C07298=1213.014,145.829,-52.403,-178.112,5.931,148.495
C07299=1213.018,145.580,-52.382,-178.114,5.929,148.495
C07300=1213.023,145.331,-52.360,-178.117,5.928,148.496
C07301=1213.027,145.082,-52.340,-178.120,5.927,148.496
C07302=1213.033,144.833,-52.319,-178.122,5.926,148.497
C07303=1213.037,144.584,-52.299,-178.125,5.924,148.497
C07304=1213.042,144.335,-52.278,-178.128,5.922,148.498
C07305=1213.047,144.085,-52.257,-178.130,5.921,148.498
C07306=1213.051,143.837,-52.236,-178.133,5.920,148.499
C07307=1213.056,143.587,-52.214,-178.135,5.919,148.499
C07308=1213.060,143.338,-52.194,-178.138,5.917,148.500
C07309=1213.066,143.089,-52.173,-178.140,5.916,148.500
C07310=1213.070,142.840,-52.153,-178.143,5.915,148.501
C07311=1213.075,142.591,-52.132,-178.145,5.914,148.501
C07312=1213.080,142.342,-52.111,-178.148,5.912,148.502
C07313=1213.084,142.093,-52.091,-178.150,5.911,148.502
C07314=1213.089,141.844,-52.070,-178.153,5.910,148.503
C07315=1213.094,141.595,-52.050,-178.156,5.909,148.503
C07316=1213.099,141.345,-52.029,-178.158,5.907,148.503
C07317=1213.103,141.096,-52.008,-178.161,5.906,148.504
C07318=1213.109,140.847,-51.987,-178.163,5.905,148.504
C07319=1213.113,140.598,-51.967,-178.167,5.903,148.505
C07320=1213.117,140.349,-51.947,-178.169,5.902,148.505
C07321=1213.123,140.100,-51.926,-178.171,5.900,148.506
C07322=1213.127,139.851,-51.905,-178.174,5.900,148.506
C07323=1213.132,139.602,-51.884,-178.177,5.898,148.507
C07324=1213.137,139.353,-51.864,-178.179,5.897,148.507
C07325=1213.141,139.104,-51.844,-178.182,5.896,148.508
C07326=1213.146,138.855,-51.823,-178.184,5.895,148.508
C07327=1213.151,138.606,-51.802,-178.187,5.893,148.509
C07328=1213.156,138.356,-51.781,-178.189,5.892,148.509
C07329=1213.160,138.107,-51.761,-178.192,5.890,148.510
C07330=1213.165,137.859,-51.740,-178.195,5.890,148.510
C07331=1213.170,137.609,-51.720,-178.197,5.888,148.511
C07332=1213.175,137.360,-51.700,-178.200,5.887,148.511
C07333=1213.179,137.111,-51.680,-178.203,5.886,148.512
C07334=1213.184,136.861,-51.659,-178.205,5.885,148.512
C07335=1213.189,136.613,-51.638,-178.208,5.883,148.513
C07336=1213.193,136.364,-51.618,-178.210,5.882,148.513
C07337=1213.198,136.114,-51.597,-178.213,5.881,148.514
C07338=1213.203,135.865,-51.577,-178.215,5.880,148.514
C07339=1213.208,135.616,-51.557,-178.218,5.878,148.514
C07340=1213.212,135.367,-51.536,-178.221,5.877,148.515
C07341=1213.217,135.118,-51.515,-178.223,5.876,148.515
C07342=1213.222,134.869,-51.495,-178.226,5.875,148.516
C07343=1213.226,134.619,-51.475,-178.229,5.873,148.516
C07344=1213.231,134.370,-51.454,-178.231,5.872,148.517
C07345=1213.237,134.122,-51.434,-178.234,5.871,148.517
C07346=1213.241,133.873,-51.414,-178.236,5.870,148.518
C07347=1213.246,133.603,-51.392,-178.239,5.868,148.518
C07348=1213.251,133.335,-51.370,-178.241,5.867,148.519
C07349=1213.256,133.066,-51.349,-178.244,5.866,148.520
C07350=1213.262,132.798,-51.326,-178.248,5.865,148.520
C07351=1213.266,132.548,-51.307,-178.250,5.864,148.521
C07352=1213.271,132.299,-51.286,-178.252,5.862,148.521
C07353=1213.275,132.050,-51.266,-178.255,5.861,148.522
C07354=1213.280,131.801,-51.246,-178.258,5.859,148.522
C07355=1213.286,131.552,-51.226,-178.260,5.859,148.523
C07356=1213.290,131.303,-51.205,-178.263,5.857,148.523
C07357=1213.295,131.054,-51.185,-178.265,5.856,148.524
C07358=1213.299,130.805,-51.165,-178.268,5.855,148.524
C07359=1213.304,130.555,-51.145,-178.270,5.854,148.524
C07360=1213.309,130.306,-51.125,-178.273,5.852,148.525
C07361=1213.314,130.057,-51.104,-178.276,5.851,148.525
C07362=1213.319,129.808,-51.085,-178.278,5.851,148.526
C07363=1213.323,129.559,-51.064,-178.281,5.849,148.526
C07364=1213.328,129.309,-51.045,-178.283,5.848,148.527
C07365=1213.333,129.060,-51.024,-178.286,5.846,148.527
C07366=1213.337,128.811,-51.005,-178.289,5.846,148.528
C07367=1213.342,128.562,-50.984,-178.291,5.844,148.528
C07368=1213.347,128.313,-50.965,-178.294,5.843,148.529
C07369=1213.352,128.064,-50.945,-178.297,5.842,148.529
C07370=1213.357,127.814,-50.924,-178.299,5.841,148.530
C07371=1213.362,127.565,-50.904,-178.301,5.840,148.531
C07372=1213.366,127.316,-50.884,-178.304,5.838,148.531
C07373=1213.371,127.067,-50.864,-178.307,5.838,148.532
C07374=1213.376,126.818,-50.845,-178.309,5.836,148.532
C07375=1213.381,126.569,-50.824,-178.312,5.835,148.533
C07376=1213.385,126.319,-50.805,-178.315,5.833,148.533
C07377=1213.390,126.070,-50.784,-178.317,5.832,148.533
C07378=1213.395,125.822,-50.765,-178.320,5.831,148.534
C07379=1213.399,125.573,-50.745,-178.322,5.830,148.534
C07380=1213.404,125.323,-50.725,-178.325,5.829,148.535
C07381=1213.409,125.073,-50.705,-178.327,5.828,148.535
C07382=1213.414,124.825,-50.685,-178.330,5.827,148.536
C07383=1213.419,124.576,-50.666,-178.333,5.825,148.536
C07384=1213.423,124.326,-50.646,-178.335,5.825,148.537
C07385=1213.428,124.077,-50.626,-178.338,5.823,148.537
C07386=1213.433,123.828,-50.606,-178.341,5.822,148.538
C07387=1213.438,123.579,-50.587,-178.343,5.821,148.539
C07388=1213.442,123.330,-50.566,-178.346,5.820,148.539
C07389=1213.447,123.080,-50.547,-178.348,5.819,148.540
C07390=1213.453,122.831,-50.527,-178.351,5.817,148.540
C07391=1213.457,122.582,-50.507,-178.353,5.817,148.541
C07392=1213.462,122.333,-50.487,-178.355,5.816,148.541
C07393=1213.466,122.083,-50.468,-178.359,5.814,148.542
C07394=1213.471,121.835,-50.448,-178.361,5.813,148.542
C07395=1213.476,121.585,-50.428,-178.364,5.812,148.543
C07396=1213.480,121.336,-50.409,-178.366,5.811,148.543
C07397=1213.486,121.087,-50.390,-178.369,5.809,148.544
C07398=1213.490,120.838,-50.369,-178.371,5.808,148.544
C07399=1213.495,120.589,-50.350,-178.374,5.808,148.545
C07400=1213.500,120.339,-50.330,-178.377,5.806,148.545
C07401=1213.505,120.090,-50.311,-178.379,5.805,148.546
C07402=1213.510,119.841,-50.291,-178.382,5.804,148.546
C07403=1213.514,119.592,-50.271,-178.385,5.803,148.547
C07404=1213.519,119.343,-50.251,-178.387,5.802,148.547
C07405=1213.523,119.094,-50.232,-178.390,5.801,148.548
C07406=1213.528,118.844,-50.213,-178.392,5.800,148.548
C07407=1213.533,118.595,-50.193,-178.395,5.798,148.549
C07408=1213.538,118.346,-50.174,-178.397,5.797,148.549
C07409=1213.544,118.097,-50.155,-178.400,5.797,148.550
C07410=1213.548,117.848,-50.134,-178.403,5.795,148.550
C07411=1213.552,117.599,-50.115,-178.405,5.794,148.551
C07412=1213.557,117.350,-50.096,-178.407,5.793,148.551
C07413=1213.562,117.100,-50.076,-178.410,5.792,148.552
C07414=1213.567,116.851,-50.056,-178.413,5.791,148.552
C07415=1213.572,116.602,-50.037,-178.416,5.789,148.553
C07416=1213.576,116.353,-50.018,-178.418,5.789,148.553
C07417=1213.581,116.103,-49.998,-178.420,5.788,148.554
C07418=1213.586,115.854,-49.979,-178.423,5.786,148.554
C07419=1213.591,115.605,-49.960,-178.426,5.786,148.555
C07420=1213.596,115.356,-49.941,-178.428,5.785,148.555
C07421=1213.600,115.106,-49.921,-178.431,5.783,148.556
C07422=1213.605,114.857,-49.902,-178.433,5.782,148.557
C07423=1213.610,114.608,-49.882,-178.436,5.781,148.557
C07424=1213.614,114.359,-49.863,-178.439,5.780,148.558
C07425=1213.620,114.110,-49.844,-178.441,5.779,148.558
C07426=1213.625,113.860,-49.824,-178.444,5.778,148.559
C07427=1213.630,113.611,-49.805,-178.446,5.777,148.559
C07428=1213.634,113.362,-49.786,-178.449,5.776,148.560
C07429=1213.639,113.113,-49.766,-178.452,5.774,148.560
C07430=1213.644,112.864,-49.747,-178.454,5.774,148.561
C07431=1213.648,112.614,-49.728,-178.456,5.773,148.561
C07432=1213.653,112.366,-49.709,-178.460,5.771,148.562
C07433=1213.658,112.116,-49.689,-178.462,5.771,148.562
C07434=1213.663,111.867,-49.670,-178.464,5.770,148.563
C07435=1213.668,111.617,-49.651,-178.467,5.768,148.563
C07436=1213.673,111.368,-49.632,-178.470,5.768,148.564
C07437=1213.677,111.119,-49.613,-178.472,5.766,148.564
C07438=1213.682,110.870,-49.594,-178.475,5.765,148.565
C07439=1213.687,110.621,-49.574,-178.477,5.764,148.566
C07440=1213.691,110.371,-49.555,-178.480,5.763,148.566
C07441=1213.697,110.123,-49.536,-178.483,5.762,148.567
C07442=1213.702,109.872,-49.517,-178.485,5.761,148.567
C07443=1213.706,109.624,-49.498,-178.488,5.760,148.568
C07444=1213.711,109.374,-49.478,-178.490,5.759,148.568
C07445=1213.716,109.126,-49.460,-178.493,5.758,148.569
C07446=1213.720,108.876,-49.440,-178.496,5.756,148.569
C07447=1213.726,108.627,-49.421,-178.498,5.756,148.570
C07448=1213.730,108.377,-49.402,-178.500,5.755,148.570
C07449=1213.735,108.129,-49.383,-178.504,5.754,148.571
C07450=1213.740,107.880,-49.364,-178.506,5.753,148.572
C07451=1213.745,107.611,-49.344,-178.508,5.752,148.572
C07452=1213.751,107.343,-49.323,-178.511,5.751,148.573
C07453=1213.756,107.073,-49.303,-178.514,5.750,148.573
C07454=1213.761,106.806,-49.283,-178.517,5.749,148.574
C07455=1213.765,106.556,-49.263,-178.519,5.748,148.574
C07456=1213.770,106.307,-49.245,-178.523,5.746,148.575
C07457=1213.775,106.058,-49.225,-178.525,5.745,148.575
C07458=1213.780,105.809,-49.207,-178.527,5.745,148.576
C07459=1213.785,105.559,-49.188,-178.530,5.743,148.576
C07460=1213.789,105.310,-49.169,-178.533,5.742,148.577
C07461=1213.795,105.061,-49.150,-178.535,5.741,148.578
C07462=1213.799,104.812,-49.132,-178.537,5.741,148.578
C07463=1213.804,104.563,-49.112,-178.541,5.739,148.579
C07464=1213.809,104.313,-49.094,-178.543,5.738,148.579
C07465=1213.814,104.064,-49.075,-178.545,5.738,148.580
C07466=1213.818,103.815,-49.056,-178.548,5.736,148.580
C07467=1213.824,103.565,-49.037,-178.551,5.735,148.581
C07468=1213.828,103.317,-49.018,-178.553,5.735,148.582
C07469=1213.833,103.066,-48.999,-178.556,5.733,148.582
C07470=1213.838,102.818,-48.981,-178.558,5.732,148.583
C07471=1213.842,102.568,-48.962,-178.561,5.731,148.583
C07472=1213.847,102.319,-48.943,-178.563,5.731,148.584
C07473=1213.852,102.070,-48.925,-178.566,5.729,148.584
C07474=1213.857,101.820,-48.905,-178.569,5.729,148.585
C07475=1213.862,101.571,-48.887,-178.571,5.728,148.585
C07476=1213.867,101.323,-48.869,-178.574,5.726,148.586
C07477=1213.872,101.072,-48.850,-178.576,5.726,148.586
C07478=1213.876,100.824,-48.831,-178.579,5.725,148.587
C07479=1213.881,100.574,-48.812,-178.581,5.724,148.587
C07480=1213.886,100.325,-48.793,-178.584,5.723,148.588
C07481=1213.891,100.076,-48.775,-178.587,5.722,148.589
C07482=1213.896,99.826,-48.756,-178.589,5.721,148.589
C07483=1213.901,99.577,-48.738,-178.592,5.719,148.590
C07484=1213.905,99.329,-48.719,-178.594,5.719,148.590
C07485=1213.910,99.078,-48.700,-178.597,5.718,148.591
C07486=1213.915,98.829,-48.682,-178.599,5.717,148.591
C07487=1213.920,98.581,-48.663,-178.602,5.716,148.592
C07488=1213.925,98.331,-48.645,-178.605,5.715,148.592
C07489=1213.929,98.082,-48.626,-178.607,5.714,148.593
C07490=1213.934,97.833,-48.608,-178.610,5.713,148.594
C07491=1213.939,97.583,-48.589,-178.612,5.712,148.594
C07492=1213.944,97.334,-48.570,-178.615,5.711,148.595
C07493=1213.949,97.085,-48.552,-178.617,5.710,148.595
C07494=1213.954,96.835,-48.534,-178.620,5.709,148.596
C07495=1213.958,96.586,-48.515,-178.623,5.708,148.596
C07496=1213.963,96.337,-48.497,-178.625,5.707,148.597
C07497=1213.968,96.088,-48.479,-178.628,5.707,148.597
C07498=1213.973,95.838,-48.459,-178.630,5.705,148.598
C07499=1213.978,95.589,-48.441,-178.633,5.704,148.599
C07500=1213.983,95.340,-48.423,-178.636,5.704,148.599
C07501=1213.988,95.091,-48.405,-178.638,5.703,148.600
C07502=1213.993,94.841,-48.385,-178.641,5.702,148.600
C07503=1213.997,94.592,-48.367,-178.644,5.701,148.601
C07504=1214.002,94.343,-48.349,-178.646,5.700,148.601
C07505=1214.007,94.094,-48.331,-178.648,5.699,148.602
C07506=1214.011,93.844,-48.312,-178.651,5.698,148.602
C07507=1214.017,93.595,-48.294,-178.654,5.697,148.603
C07508=1214.022,93.346,-48.276,-178.656,5.696,148.604
C07509=1214.027,93.097,-48.258,-178.658,5.696,148.604
C07510=1214.031,92.847,-48.240,-178.662,5.694,148.605
C07511=1214.036,92.598,-48.221,-178.664,5.694,148.605
C07512=1214.041,92.349,-48.202,-178.666,5.693,148.606
C07513=1214.046,92.099,-48.184,-178.669,5.692,148.606
C07514=1214.051,91.850,-48.166,-178.672,5.690,148.607
C07515=1214.055,91.600,-48.148,-178.674,5.690,148.608
C07516=1214.060,91.351,-48.130,-178.677,5.689,148.608
C07517=1214.065,91.102,-48.112,-178.679,5.688,148.609
C07518=1214.070,90.853,-48.093,-178.682,5.687,148.609
C07519=1214.075,90.603,-48.074,-178.685,5.686,148.610
C07520=1214.080,90.354,-48.056,-178.687,5.685,148.610
C07521=1214.085,90.105,-48.038,-178.690,5.685,148.611
C07522=1214.090,89.856,-48.020,-178.692,5.684,148.612
C07523=1214.095,89.607,-48.002,-178.695,5.682,148.612
C07524=1214.099,89.357,-47.984,-178.698,5.682,148.613
C07525=1214.104,89.108,-47.966,-178.700,5.681,148.613
C07526=1214.109,88.858,-47.948,-178.702,5.680,148.614
C07527=1214.114,88.609,-47.930,-178.706,5.679,148.614
C07528=1214.119,88.360,-47.912,-178.708,5.678,148.615
C07529=1214.123,88.111,-47.894,-178.710,5.677,148.615
C07530=1214.128,87.861,-47.876,-178.713,5.677,148.616
C07531=1214.133,87.611,-47.857,-178.715,5.676,148.617
C07532=1214.138,87.362,-47.839,-178.718,5.674,148.617
C07533=1214.143,87.113,-47.821,-178.721,5.674,148.618
C07534=1214.148,86.864,-47.803,-178.723,5.673,148.618
C07535=1214.153,86.615,-47.785,-178.726,5.672,148.619
C07536=1214.158,86.366,-47.767,-178.728,5.672,148.620
C07537=1214.163,86.116,-47.749,-178.731,5.670,148.620
C07538=1214.167,85.867,-47.731,-178.734,5.669,148.621
C07539=1214.172,85.617,-47.713,-178.736,5.669,148.621
C07540=1214.177,85.368,-47.695,-178.738,5.668,148.622
C07541=1214.182,85.119,-47.677,-178.741,5.667,148.622
C07542=1214.187,84.869,-47.660,-178.744,5.666,148.623
C07543=1214.192,84.620,-47.642,-178.746,5.665,148.623
C07544=1214.197,84.371,-47.624,-178.749,5.664,148.624
C07545=1214.202,84.122,-47.606,-178.752,5.664,148.625
C07546=1214.207,83.873,-47.588,-178.754,5.663,148.625
C07547=1214.210,83.623,-47.570,-178.757,5.661,148.626
C07548=1214.215,83.374,-47.552,-178.759,5.661,148.626
C07549=1214.220,83.125,-47.534,-178.762,5.660,148.627
C07550=1214.225,82.875,-47.517,-178.764,5.659,148.628
C07551=1214.230,82.626,-47.499,-178.767,5.659,148.628
C07552=1214.235,82.376,-47.481,-178.770,5.657,148.629
C07553=1214.240,82.127,-47.463,-178.772,5.656,148.629
C07554=1214.245,81.878,-47.445,-178.775,5.656,148.630
C07555=1214.250,81.609,-47.426,-178.777,5.655,148.631
C07556=1214.256,81.341,-47.407,-178.781,5.654,148.631
C07557=1214.261,81.073,-47.387,-178.783,5.653,148.632
C07558=1214.266,80.804,-47.369,-178.785,5.652,148.632
C07559=1214.271,80.555,-47.351,-178.788,5.652,148.633
C07560=1214.276,80.305,-47.333,-178.791,5.650,148.634
C07561=1214.281,80.056,-47.316,-178.793,5.649,148.634
C07562=1214.285,79.807,-47.298,-178.796,5.649,148.635
C07563=1214.290,79.558,-47.280,-178.799,5.648,148.635
C07564=1214.295,79.308,-47.263,-178.801,5.647,148.636
C07565=1214.300,79.059,-47.245,-178.803,5.647,148.636
C07566=1214.305,78.810,-47.227,-178.807,5.645,148.637
C07567=1214.310,78.560,-47.210,-178.809,5.645,148.638
C07568=1214.315,78.311,-47.192,-178.811,5.644,148.638
C07569=1214.319,78.062,-47.174,-178.814,5.643,148.639
C07570=1214.325,77.812,-47.157,-178.817,5.643,148.640
C07571=1214.330,77.563,-47.139,-178.819,5.642,148.640
C07572=1214.335,77.314,-47.121,-178.822,5.640,148.641
C07573=1214.339,77.064,-47.104,-178.825,5.640,148.641
C07574=1214.344,76.815,-47.086,-178.827,5.639,148.642
C07575=1214.349,76.566,-47.069,-178.829,5.638,148.642
C07576=1214.354,76.316,-47.051,-178.832,5.638,148.643
C07577=1214.358,76.067,-47.034,-178.835,5.637,148.644
C07578=1214.364,75.818,-47.017,-178.837,5.635,148.644
C07579=1214.369,75.569,-46.999,-178.840,5.635,148.645
C07580=1214.374,75.319,-46.982,-178.843,5.634,148.645
C07581=1214.378,75.070,-46.964,-178.845,5.633,148.646
C07582=1214.384,74.820,-46.947,-178.847,5.633,148.646
C07583=1214.388,74.571,-46.929,-178.850,5.632,148.647
C07584=1214.394,74.321,-46.912,-178.852,5.631,148.648
C07585=1214.398,74.072,-46.894,-178.855,5.630,148.648
C07586=1214.403,73.823,-46.877,-178.858,5.629,148.649
C07587=1214.408,73.573,-46.859,-178.861,5.629,148.650
C07588=1214.412,73.324,-46.843,-178.863,5.628,148.650
C07589=1214.417,73.075,-46.825,-178.865,5.627,148.651
C07590=1214.423,72.825,-46.807,-178.868,5.627,148.651
C07591=1214.427,72.576,-46.790,-178.870,5.626,148.652
C07592=1214.432,72.326,-46.773,-178.873,5.625,148.652
C07593=1214.438,72.078,-46.755,-178.876,5.624,148.653
C07594=1214.442,71.828,-46.738,-178.879,5.623,148.654
C07595=1214.447,71.579,-46.720,-178.881,5.622,148.654
C07596=1214.452,71.329,-46.703,-178.883,5.622,148.655
C07597=1214.457,71.080,-46.686,-178.886,5.621,148.655
C07598=1214.462,70.831,-46.668,-178.889,5.620,148.656
C07599=1214.467,70.581,-46.651,-178.891,5.620,148.657
C07600=1214.471,70.332,-46.634,-178.893,5.619,148.657
C07601=1214.477,70.083,-46.617,-178.897,5.618,148.658
C07602=1214.481,69.834,-46.600,-178.899,5.617,148.658
C07603=1214.486,69.584,-46.582,-178.901,5.616,148.659
C07604=1214.491,69.335,-46.565,-178.904,5.616,148.660
C07605=1214.496,69.085,-46.548,-178.907,5.615,148.660
C07606=1214.501,68.836,-46.530,-178.909,5.614,148.661
C07607=1214.505,68.586,-46.514,-178.911,5.613,148.661
C07608=1214.511,68.337,-46.497,-178.914,5.613,148.662
C07609=1214.516,68.088,-46.479,-178.917,5.612,148.663
C07610=1214.520,67.839,-46.462,-178.919,5.611,148.663
C07611=1214.526,67.589,-46.445,-178.922,5.610,148.664
C07612=1214.530,67.339,-46.428,-178.925,5.609,148.664
C07613=1214.535,67.090,-46.410,-178.927,5.609,148.665
C07614=1214.540,66.841,-46.394,-178.929,5.608,148.666
C07615=1214.545,66.592,-46.377,-178.932,5.607,148.666
C07616=1214.550,66.342,-46.360,-178.935,5.607,148.667
C07617=1214.555,66.093,-46.342,-178.937,5.606,148.668
C07618=1214.559,65.844,-46.325,-178.939,5.605,148.668
C07619=1214.564,65.594,-46.308,-178.942,5.605,148.669
C07620=1214.569,65.345,-46.292,-178.945,5.603,148.669
C07621=1214.575,65.095,-46.274,-178.948,5.603,148.670
C07622=1214.579,64.846,-46.257,-178.950,5.602,148.670
C07623=1214.584,64.596,-46.240,-178.953,5.601,148.671
C07624=1214.589,64.348,-46.224,-178.955,5.601,148.672
C07625=1214.594,64.098,-46.206,-178.958,5.600,148.672
C07626=1214.599,63.848,-46.190,-178.960,5.599,148.673
C07627=1214.604,63.599,-46.172,-178.963,5.599,148.673
C07628=1214.608,63.350,-46.155,-178.965,5.598,148.674
C07629=1214.614,63.101,-46.138,-178.968,5.598,148.675
C07630=1214.619,62.851,-46.121,-178.970,5.597,148.675
C07631=1214.623,62.602,-46.105,-178.973,5.596,148.676
C07632=1214.628,62.352,-46.087,-178.976,5.595,148.677
C07633=1214.633,62.103,-46.071,-178.979,5.594,148.677
C07634=1214.639,61.853,-46.054,-178.981,5.593,148.678
C07635=1214.643,61.604,-46.037,-178.983,5.593,148.678
C07636=1214.648,61.355,-46.021,-178.986,5.592,148.679
C07637=1214.653,61.105,-46.004,-178.989,5.592,148.680
C07638=1214.658,60.856,-45.987,-178.991,5.591,148.680
C07639=1214.663,60.606,-45.970,-178.993,5.590,148.681
C07640=1214.668,60.357,-45.953,-178.996,5.590,148.681
C07641=1214.673,60.108,-45.937,-178.999,5.589,148.682
C07642=1214.678,59.858,-45.919,-179.001,5.588,148.682
C07643=1214.682,59.608,-45.903,-179.003,5.588,148.683
C07644=1214.687,59.360,-45.887,-179.006,5.587,148.684
C07645=1214.693,59.110,-45.869,-179.009,5.586,148.684
C07646=1214.697,58.860,-45.853,-179.012,5.585,148.685
C07647=1214.702,58.612,-45.836,-179.014,5.584,148.686
C07648=1214.707,58.362,-45.819,-179.017,5.584,148.686
C07649=1214.712,58.112,-45.802,-179.019,5.583,148.687
C07650=1214.717,57.864,-45.786,-179.022,5.582,148.688
C07651=1214.722,57.614,-45.769,-179.024,5.581,148.688
C07652=1214.727,57.364,-45.752,-179.027,5.581,148.689
C07653=1214.732,57.115,-45.736,-179.029,5.580,148.689
C07654=1214.737,56.866,-45.719,-179.032,5.580,148.690
C07655=1214.741,56.616,-45.702,-179.035,5.579,148.691
C07656=1214.746,56.367,-45.686,-179.037,5.578,148.691
C07657=1214.752,56.118,-45.668,-179.039,5.578,148.692
C07658=1214.757,55.867,-45.652,-179.042,5.577,148.692
C07659=1214.762,55.600,-45.635,-179.045,5.577,148.693
C07660=1214.767,55.332,-45.617,-179.048,5.575,148.694
C07661=1214.773,55.062,-45.599,-179.050,5.575,148.694
C07662=1214.778,54.794,-45.581,-179.053,5.574,148.695
C07663=1214.782,54.545,-45.564,-179.056,5.574,148.696
C07664=1214.788,54.295,-45.547,-179.058,5.573,148.696
C07665=1214.793,54.046,-45.531,-179.061,5.572,148.697
C07666=1214.798,53.796,-45.515,-179.063,5.572,148.698
C07667=1214.803,53.547,-45.499,-179.066,5.571,148.698
C07668=1214.807,53.298,-45.482,-179.068,5.570,148.699
C07669=1214.812,53.048,-45.465,-179.071,5.570,148.699
C07670=1214.817,52.799,-45.448,-179.073,5.569,148.700
C07671=1214.822,52.549,-45.432,-179.076,5.568,148.701
C07672=1214.827,52.301,-45.416,-179.078,5.568,148.701
C07673=1214.832,52.051,-45.400,-179.081,5.567,148.702
C07674=1214.837,51.801,-45.382,-179.083,5.566,148.702
C07675=1214.842,51.552,-45.367,-179.086,5.566,148.703
C07676=1214.847,51.302,-45.350,-179.089,5.565,148.704
C07677=1214.852,51.054,-45.334,-179.091,5.565,148.704
C07678=1214.857,50.803,-45.318,-179.094,5.564,148.705
C07679=1214.862,50.555,-45.301,-179.096,5.563,148.706
C07680=1214.866,50.305,-45.285,-179.099,5.563,148.706
C07681=1214.872,50.055,-45.268,-179.101,5.562,148.707
C07682=1214.877,49.806,-45.252,-179.104,5.562,148.708
C07683=1214.881,49.557,-45.235,-179.106,5.561,148.708
C07684=1214.887,49.307,-45.220,-179.109,5.559,148.709
C07685=1214.891,49.058,-45.203,-179.112,5.559,148.709
C07686=1214.896,48.809,-45.187,-179.114,5.558,148.710
C07687=1214.901,48.559,-45.171,-179.117,5.558,148.711
C07688=1214.906,48.310,-45.154,-179.120,5.557,148.711
C07689=1214.911,48.060,-45.138,-179.122,5.557,148.712
C07690=1214.916,47.811,-45.122,-179.125,5.556,148.712
C07691=1214.920,47.562,-45.105,-179.127,5.555,148.713
C07692=1214.927,47.312,-45.089,-179.130,5.555,148.714
C07693=1214.931,47.062,-45.073,-179.132,5.554,148.714
C07694=1214.936,46.813,-45.057,-179.135,5.554,148.715
C07695=1214.941,46.564,-45.040,-179.137,5.553,148.716
C07696=1214.946,46.315,-45.024,-179.140,5.552,148.716
C07697=1214.951,46.065,-45.008,-179.143,5.552,148.717
C07698=1214.956,45.816,-44.992,-179.145,5.551,148.718
C07699=1214.961,45.566,-44.976,-179.148,5.550,148.718
C07700=1214.966,45.317,-44.960,-179.150,5.550,148.719
C07701=1214.971,45.067,-44.944,-179.153,5.549,148.719
C07702=1214.976,44.818,-44.927,-179.155,5.548,148.720
C07703=1214.980,44.568,-44.911,-179.158,5.548,148.721
C07704=1214.985,44.319,-44.895,-179.161,5.547,148.721
C07705=1214.990,44.069,-44.879,-179.163,5.548,148.722
C07706=1214.996,43.820,-44.864,-179.165,5.547,148.723
C07707=1215.000,43.570,-44.847,-179.167,5.546,148.723
C07708=1215.006,43.321,-44.831,-179.170,5.546,148.724
C07709=1215.010,43.071,-44.815,-179.173,5.545,148.725
C07710=1215.015,42.822,-44.799,-179.175,5.544,148.725
C07711=1215.020,42.573,-44.783,-179.178,5.544,148.726
C07712=1215.025,42.323,-44.767,-179.180,5.543,148.726
C07713=1215.031,42.074,-44.751,-179.183,5.542,148.727
C07714=1215.035,41.824,-44.734,-179.185,5.542,148.728
C07715=1215.040,41.575,-44.719,-179.188,5.541,148.728
C07716=1215.044,41.326,-44.703,-179.191,5.541,148.729
C07717=1215.050,41.076,-44.687,-179.193,5.540,148.730
C07718=1215.055,40.827,-44.672,-179.195,5.539,148.730
C07719=1215.060,40.577,-44.655,-179.198,5.539,148.731
C07720=1215.065,40.328,-44.639,-179.201,5.538,148.731
C07721=1215.070,40.078,-44.623,-179.203,5.538,148.732
C07722=1215.075,39.829,-44.607,-179.206,5.537,148.733
C07723=1215.080,39.580,-44.592,-179.209,5.537,148.734
C07724=1215.085,39.329,-44.576,-179.211,5.536,148.734
C07725=1215.089,39.081,-44.560,-179.213,5.535,148.735
C07726=1215.094,38.831,-44.544,-179.216,5.535,148.735
C07727=1215.099,38.582,-44.528,-179.219,5.534,148.736
C07728=1215.105,38.332,-44.513,-179.221,5.534,148.737
C07729=1215.109,38.083,-44.496,-179.224,5.533,148.737
C07730=1215.115,37.833,-44.480,-179.226,5.532,148.738
C07731=1215.120,37.584,-44.465,-179.229,5.532,148.738
C07732=1215.124,37.335,-44.449,-179.231,5.531,148.739
C07733=1215.129,37.085,-44.433,-179.234,5.531,148.740
C07734=1215.135,36.836,-44.418,-179.237,5.530,148.740
C07735=1215.139,36.586,-44.402,-179.239,5.529,148.741
C07736=1215.145,36.336,-44.386,-179.242,5.529,148.742
C07737=1215.149,36.088,-44.370,-179.244,5.529,148.742
C07738=1215.154,35.838,-44.354,-179.246,5.528,148.743
C07739=1215.159,35.588,-44.339,-179.249,5.528,148.744
C07740=1215.165,35.339,-44.323,-179.251,5.527,148.744
C07741=1215.169,35.089,-44.307,-179.254,5.527,148.745
C07742=1215.174,34.840,-44.292,-179.257,5.526,148.746
C07743=1215.179,34.591,-44.276,-179.259,5.525,148.746
C07744=1215.184,34.341,-44.260,-179.262,5.525,148.747
C07745=1215.189,34.091,-44.244,-179.264,5.524,148.747
C07746=1215.194,33.842,-44.229,-179.267,5.524,148.748
C07747=1215.199,33.592,-44.214,-179.269,5.523,148.749
C07748=1215.204,33.343,-44.198,-179.272,5.523,148.749
C07749=1215.210,33.093,-44.182,-179.275,5.522,148.750
C07750=1215.214,32.844,-44.167,-179.277,5.521,148.751
C07751=1215.219,32.595,-44.151,-179.280,5.521,148.751
C07752=1215.224,32.345,-44.135,-179.282,5.520,148.752
C07753=1215.229,32.096,-44.120,-179.284,5.520,148.753
C07754=1215.234,31.846,-44.104,-179.287,5.520,148.753
C07755=1215.239,31.597,-44.089,-179.290,5.519,148.754
C07756=1215.244,31.347,-44.073,-179.292,5.519,148.755
C07757=1215.248,31.098,-44.058,-179.294,5.518,148.755
C07758=1215.254,30.848,-44.042,-179.297,5.517,148.756
C07759=1215.259,30.599,-44.026,-179.300,5.517,148.756
C07760=1215.264,30.350,-44.011,-179.302,5.516,148.757
C07761=1215.269,30.100,-43.996,-179.305,5.516,148.758
C07762=1215.274,29.850,-43.980,-179.308,5.515,148.758
C07763=1215.279,29.582,-43.964,-179.310,5.515,148.759
C07764=1215.285,29.313,-43.947,-179.313,5.514,148.760
C07765=1215.290,29.045,-43.930,-179.316,5.513,148.761
C07766=1215.295,28.776,-43.914,-179.318,5.513,148.761
C07767=1215.300,28.527,-43.898,-179.321,5.512,148.762
C07768=1215.306,28.276,-43.883,-179.323,5.512,148.763
C07769=1215.310,28.027,-43.868,-179.326,5.511,148.763
C07770=1215.316,27.778,-43.852,-179.329,5.511,148.764
C07771=1215.320,27.529,-43.837,-179.331,5.510,148.764
C07772=1215.325,27.279,-43.821,-179.334,5.509,148.765
C07773=1215.330,27.029,-43.806,-179.336,5.510,148.766
C07774=1215.335,26.780,-43.791,-179.338,5.509,148.766
C07775=1215.340,26.531,-43.775,-179.341,5.509,148.767
C07776=1215.345,26.282,-43.760,-179.344,5.508,148.768
C07777=1215.350,26.032,-43.745,-179.346,5.508,148.768
C07778=1215.356,25.781,-43.729,-179.349,5.507,148.769
C07779=1215.360,25.532,-43.714,-179.351,5.506,148.770
C07780=1215.366,25.283,-43.699,-179.354,5.506,148.770
C07781=1215.370,25.034,-43.684,-179.356,5.505,148.771
C07782=1215.376,24.784,-43.668,-179.359,5.505,148.772
C07783=1215.380,24.535,-43.653,-179.361,5.505,148.772
C07784=1215.385,24.285,-43.638,-179.364,5.504,148.773
C07785=1215.390,24.036,-43.623,-179.366,5.504,148.774
C07786=1215.395,23.786,-43.607,-179.369,5.503,148.774
C07787=1215.400,23.537,-43.592,-179.371,5.502,148.775
C07788=1215.405,23.288,-43.577,-179.374,5.502,148.775
C07789=1215.410,23.038,-43.563,-179.376,5.501,148.776
C07790=1215.415,22.788,-43.547,-179.379,5.501,148.777
C07791=1215.420,22.539,-43.532,-179.382,5.500,148.777
C07792=1215.425,22.289,-43.516,-179.384,5.500,148.778
C07793=1215.430,22.040,-43.502,-179.386,5.500,148.779
C07794=1215.436,21.790,-43.486,-179.389,5.499,148.780
C07795=1215.440,21.541,-43.471,-179.392,5.499,148.780
C07796=1215.446,21.292,-43.456,-179.394,5.498,148.781
C07797=1215.451,21.042,-43.441,-179.396,5.497,148.781
C07798=1215.455,20.792,-43.425,-179.399,5.497,148.782
C07799=1215.460,20.543,-43.410,-179.402,5.496,148.783
C07800=1215.465,20.293,-43.396,-179.404,5.496,148.783
C07801=1215.470,20.044,-43.381,-179.406,5.496,148.784
C07802=1215.475,19.795,-43.366,-179.409,5.496,148.785
C07803=1215.481,19.545,-43.351,-179.412,5.495,148.785
C07804=1215.485,19.296,-43.336,-179.414,5.495,148.786
C07805=1215.491,19.046,-43.320,-179.417,5.494,148.787
C07806=1215.496,18.796,-43.306,-179.419,5.493,148.787
C07807=1215.500,18.547,-43.291,-179.422,5.493,148.788
C07808=1215.506,18.298,-43.275,-179.425,5.492,148.789
C07809=1215.510,18.048,-43.261,-179.427,5.492,148.789
C07810=1215.515,17.798,-43.246,-179.429,5.492,148.790
C07811=1215.520,17.548,-43.231,-179.432,5.491,148.791
C07812=1215.525,17.299,-43.216,-179.435,5.491,148.791
C07813=1215.531,17.049,-43.201,-179.437,5.490,148.792
C07814=1215.535,16.800,-43.186,-179.439,5.489,148.792
C07815=1215.540,16.551,-43.171,-179.442,5.489,148.793
C07816=1215.546,16.301,-43.156,-179.444,5.489,148.794
C07817=1215.550,16.052,-43.141,-179.447,5.489,148.795
C07818=1215.555,15.802,-43.127,-179.449,5.488,148.795
C07819=1215.561,15.553,-43.111,-179.452,5.488,148.796
C07820=1215.566,15.303,-43.097,-179.455,5.487,148.797
C07821=1215.570,15.054,-43.082,-179.457,5.487,148.797
C07822=1215.576,14.804,-43.067,-179.460,5.486,148.798
C07823=1215.581,14.555,-43.052,-179.462,5.486,148.799
C07824=1215.586,14.305,-43.038,-179.464,5.485,148.799
C07825=1215.590,14.056,-43.023,-179.467,5.485,148.800
C07826=1215.596,13.806,-43.008,-179.469,5.484,148.800
C07827=1215.601,13.557,-42.993,-179.472,5.484,148.801
C07828=1215.606,13.307,-42.979,-179.475,5.483,148.802
C07829=1215.611,13.058,-42.963,-179.477,5.483,148.803
C07830=1215.616,12.808,-42.949,-179.479,5.483,148.803
C07831=1215.621,12.559,-42.934,-179.482,5.483,148.804
C07832=1215.625,12.309,-42.919,-179.485,5.482,148.805
C07833=1215.631,12.059,-42.905,-179.487,5.482,148.805
C07834=1215.636,11.810,-42.890,-179.490,5.481,148.806
C07835=1215.641,11.561,-42.875,-179.492,5.480,148.806
C07836=1215.645,11.312,-42.860,-179.494,5.480,148.807
C07837=1215.651,11.061,-42.845,-179.497,5.480,148.808
C07838=1215.656,10.812,-42.831,-179.500,5.479,148.808
C07839=1215.661,10.563,-42.816,-179.502,5.479,148.809
C07840=1215.666,10.313,-42.802,-179.505,5.478,148.810
C07841=1215.671,10.063,-42.788,-179.508,5.478,148.811
C07842=1215.676,9.814,-42.772,-179.510,5.478,148.811
C07843=1215.681,9.564,-42.758,-179.512,5.478,148.812
C07844=1215.686,9.314,-42.743,-179.515,5.477,148.813
C07845=1215.691,9.065,-42.728,-179.517,5.476,148.813
C07846=1215.696,8.816,-42.715,-179.520,5.476,148.814
C07847=1215.702,8.566,-42.700,-179.522,5.475,148.814
C07848=1215.706,8.317,-42.685,-179.524,5.475,148.815
C07849=1215.711,8.068,-42.670,-179.527,5.475,148.816
C07850=1215.716,7.818,-42.656,-179.530,5.474,148.816
C07851=1215.721,7.568,-42.642,-179.532,5.474,148.817
C07852=1215.726,7.319,-42.627,-179.535,5.473,148.818
C07853=1215.731,7.069,-42.613,-179.538,5.473,148.819
C07854=1215.737,6.819,-42.598,-179.540,5.473,148.819
C07855=1215.742,6.570,-42.583,-179.542,5.473,148.820
C07856=1215.746,6.320,-42.568,-179.545,5.472,148.821
C07857=1215.752,6.071,-42.555,-179.547,5.471,148.821
C07858=1215.757,5.822,-42.540,-179.550,5.471,148.822
C07859=1215.762,5.572,-42.526,-179.552,5.471,148.822
C07860=1215.766,5.323,-42.511,-179.555,5.471,148.823
C07861=1215.771,5.073,-42.497,-179.557,5.470,148.824
C07862=1215.776,4.824,-42.482,-179.560,5.470,148.824
C07863=1215.781,4.574,-42.468,-179.563,5.469,148.825
C07864=1215.787,4.324,-42.453,-179.565,5.468,148.826
C07865=1215.792,4.075,-42.439,-179.567,5.469,148.827
C07866=1215.797,3.826,-42.424,-179.570,5.468,148.827
C07867=1215.803,3.556,-42.409,-179.573,5.468,148.828
C07868=1215.808,3.287,-42.394,-179.575,5.467,148.829
C07869=1215.813,3.018,-42.379,-179.578,5.467,148.829
C07870=1215.818,2.749,-42.363,-179.581,5.466,148.830
C07871=1215.823,2.500,-42.349,-179.583,5.466,148.831
C07872=1215.828,2.250,-42.334,-179.586,5.465,148.831
C07873=1215.834,2.001,-42.321,-179.588,5.465,148.832
C07874=1215.839,1.751,-42.306,-179.591,5.465,148.833
C07875=1215.844,1.501,-42.292,-179.593,5.464,148.833
C07876=1215.848,1.252,-42.277,-179.596,5.464,148.834
C07877=1215.853,1.003,-42.263,-179.599,5.463,148.835
C07878=1215.859,0.754,-42.249,-179.601,5.464,148.835
C07879=1215.864,0.504,-42.235,-179.603,5.463,148.836
C07880=1215.869,0.254,-42.220,-179.606,5.463,148.837
C07881=1215.874,0.004,-42.206,-179.608,5.462,148.837
C07882=1215.879,-0.245,-42.192,-179.610,5.462,148.838
C07883=1215.884,-0.494,-42.178,-179.613,5.462,148.839
C07884=1215.889,-0.744,-42.163,-179.616,5.461,148.839
C07885=1215.894,-0.994,-42.149,-179.618,5.461,148.840
C07886=1215.899,-1.243,-42.135,-179.621,5.460,148.841
C07887=1215.904,-1.493,-42.121,-179.623,5.460,148.841
C07888=1215.910,-1.742,-42.107,-179.626,5.460,148.842
C07889=1215.914,-1.992,-42.092,-179.628,5.459,148.843
C07890=1215.919,-2.242,-42.078,-179.631,5.459,148.844
C07891=1215.924,-2.491,-42.064,-179.634,5.458,148.844
C07892=1215.930,-2.740,-42.050,-179.636,5.459,148.845
C07893=1215.935,-2.990,-42.036,-179.638,5.458,148.846
C07894=1215.940,-3.240,-42.021,-179.641,5.458,148.846
C07895=1215.944,-3.490,-42.008,-179.643,5.457,148.847
C07896=1215.950,-3.739,-41.995,-179.645,5.457,148.847
C07897=1215.955,-3.988,-41.980,-179.648,5.457,148.848
C07898=1215.960,-4.238,-41.966,-179.650,5.456,148.849
C07899=1215.965,-4.488,-41.952,-179.653,5.456,148.849
C07900=1215.970,-4.737,-41.938,-179.656,5.455,148.850
C07901=1215.975,-4.987,-41.924,-179.658,5.455,148.851
C07902=1215.980,-5.236,-41.909,-179.660,5.455,148.852
C07903=1215.984,-5.486,-41.896,-179.663,5.454,148.852
C07904=1215.990,-5.735,-41.882,-179.666,5.454,148.853
C07905=1215.995,-5.985,-41.868,-179.668,5.454,148.854
C07906=1216.000,-6.235,-41.854,-179.671,5.454,148.854
C07907=1216.006,-6.484,-41.840,-179.673,5.453,148.855
C07908=1216.011,-6.733,-41.826,-179.676,5.453,148.856
C07909=1216.015,-6.983,-41.812,-179.678,5.453,148.856
C07910=1216.020,-7.233,-41.798,-179.680,5.452,148.857
C07911=1216.026,-7.482,-41.785,-179.683,5.452,148.858
C07912=1216.031,-7.732,-41.770,-179.685,5.451,148.858
C07913=1216.036,-7.982,-41.756,-179.688,5.451,148.859
C07914=1216.041,-8.230,-41.743,-179.690,5.451,148.860
C07915=1216.046,-8.481,-41.729,-179.693,5.450,148.860
C07916=1216.051,-8.730,-41.715,-179.695,5.450,148.861
C07917=1216.056,-8.979,-41.701,-179.698,5.449,148.862
C07918=1216.061,-9.229,-41.687,-179.700,5.450,148.862
C07919=1216.066,-9.479,-41.674,-179.703,5.449,148.863
C07920=1216.071,-9.728,-41.660,-179.705,5.449,148.864
C07921=1216.076,-9.978,-41.645,-179.708,5.448,148.864
C07922=1216.082,-10.228,-41.632,-179.710,5.448,148.865
C07923=1216.086,-10.477,-41.619,-179.713,5.448,148.866
C07924=1216.091,-10.727,-41.604,-179.716,5.447,148.867
C07925=1216.096,-10.976,-41.590,-179.718,5.447,148.867
C07926=1216.102,-11.226,-41.577,-179.720,5.447,148.868
C07927=1216.106,-11.475,-41.563,-179.722,5.446,148.868
C07928=1216.112,-11.724,-41.549,-179.725,5.446,148.869
C07929=1216.117,-11.975,-41.536,-179.728,5.445,148.870
C07930=1216.121,-12.224,-41.522,-179.730,5.446,148.870
C07931=1216.127,-12.473,-41.508,-179.732,5.445,148.871
C07932=1216.132,-12.723,-41.495,-179.735,5.445,148.872
C07933=1216.136,-12.973,-41.481,-179.738,5.444,148.873
C07934=1216.142,-13.222,-41.468,-179.740,5.445,148.873
C07935=1216.147,-13.472,-41.453,-179.743,5.444,148.874
C07936=1216.152,-13.721,-41.440,-179.745,5.444,148.875
C07937=1216.157,-13.971,-41.426,-179.748,5.443,148.875
C07938=1216.162,-14.221,-41.412,-179.750,5.443,148.876
C07939=1216.167,-14.470,-41.400,-179.753,5.443,148.877
C07940=1216.172,-14.720,-41.385,-179.755,5.442,148.877
C07941=1216.178,-14.969,-41.371,-179.757,5.443,148.878
C07942=1216.182,-15.219,-41.358,-179.760,5.442,148.879
C07943=1216.187,-15.469,-41.344,-179.762,5.441,148.879
C07944=1216.193,-15.718,-41.331,-179.765,5.441,148.880
C07945=1216.197,-15.968,-41.317,-179.767,5.441,148.881
C07946=1216.203,-16.217,-41.304,-179.770,5.441,148.881
C07947=1216.208,-16.467,-41.290,-179.772,5.440,148.882
C07948=1216.213,-16.716,-41.277,-179.775,5.440,148.883
C07949=1216.218,-16.966,-41.263,-179.777,5.440,148.883
C07950=1216.223,-17.215,-41.250,-179.780,5.439,148.884
C07951=1216.228,-17.465,-41.236,-179.782,5.439,148.885
C07952=1216.234,-17.715,-41.223,-179.785,5.438,148.885
C07953=1216.238,-17.964,-41.209,-179.787,5.439,148.886
C07954=1216.244,-18.214,-41.196,-179.790,5.438,148.887
C07955=1216.249,-18.463,-41.182,-179.792,5.438,148.888
C07956=1216.254,-18.713,-41.169,-179.794,5.438,148.888
C07957=1216.259,-18.962,-41.155,-179.797,5.438,148.889
C07958=1216.264,-19.212,-41.142,-179.800,5.437,148.890
C07959=1216.270,-19.462,-41.129,-179.802,5.437,148.890
C07960=1216.274,-19.711,-41.115,-179.804,5.437,148.891
C07961=1216.280,-19.961,-41.102,-179.807,5.436,148.892
C07962=1216.284,-20.210,-41.088,-179.809,5.436,148.892
C07963=1216.290,-20.460,-41.075,-179.811,5.436,148.893
C07964=1216.294,-20.710,-41.062,-179.814,5.435,148.894
C07965=1216.300,-20.959,-41.048,-179.817,5.435,148.894
C07966=1216.305,-21.209,-41.035,-179.819,5.434,148.895
C07967=1216.310,-21.458,-41.021,-179.821,5.435,148.896
C07968=1216.315,-21.708,-41.008,-179.824,5.434,148.896
C07969=1216.320,-21.958,-40.995,-179.827,5.434,148.897
C07970=1216.325,-22.207,-40.981,-179.829,5.434,148.898
C07971=1216.331,-22.477,-40.967,-179.831,5.434,148.898
C07972=1216.336,-22.746,-40.952,-179.834,5.433,148.899
C07973=1216.341,-23.016,-40.939,-179.837,5.433,148.900
C07974=1216.347,-23.285,-40.924,-179.840,5.432,148.901
C07975=1216.352,-23.534,-40.911,-179.842,5.433,148.901
C07976=1216.358,-23.784,-40.898,-179.845,5.432,148.902
C07977=1216.362,-24.033,-40.884,-179.847,5.432,148.903
C07978=1216.368,-24.283,-40.871,-179.850,5.431,148.904
C07979=1216.372,-24.533,-40.858,-179.852,5.431,148.904
C07980=1216.378,-24.783,-40.845,-179.854,5.431,148.905
C07981=1216.383,-25.032,-40.831,-179.857,5.430,148.905
C07982=1216.388,-25.281,-40.819,-179.859,5.431,148.906
C07983=1216.393,-25.532,-40.805,-179.862,5.430,148.907
C07984=1216.398,-25.781,-40.792,-179.864,5.430,148.908
C07985=1216.403,-26.031,-40.778,-179.866,5.430,148.908
C07986=1216.408,-26.280,-40.766,-179.869,5.429,148.909
C07987=1216.413,-26.529,-40.753,-179.872,5.429,148.910
C07988=1216.419,-26.780,-40.739,-179.874,5.428,148.910
C07989=1216.423,-27.028,-40.726,-179.876,5.429,148.911
C07990=1216.429,-27.279,-40.713,-179.879,5.428,148.912
C07991=1216.434,-27.528,-40.700,-179.882,5.428,148.912
C07992=1216.439,-27.777,-40.687,-179.884,5.428,148.913
C07993=1216.444,-28.028,-40.674,-179.886,5.428,148.914
C07994=1216.449,-28.277,-40.661,-179.889,5.427,148.914
C07995=1216.453,-28.526,-40.647,-179.891,5.427,148.915
C07996=1216.459,-28.776,-40.634,-179.894,5.427,148.916
C07997=1216.464,-29.025,-40.622,-179.897,5.427,148.917
C07998=1216.469,-29.275,-40.609,-179.898,5.426,148.917
C07999=1216.475,-29.525,-40.596,-179.901,5.426,148.918
C08000=1216.479,-29.775,-40.583,-179.903,5.425,148.918
C08001=1216.484,-30.024,-40.570,-179.906,5.426,148.919
C08002=1216.490,-30.274,-40.557,-179.908,5.425,148.920
C08003=1216.495,-30.523,-40.543,-179.911,5.425,148.921
C08004=1216.500,-30.773,-40.530,-179.914,5.424,148.921
C08005=1216.506,-31.022,-40.517,-179.916,5.425,148.922
C08006=1216.510,-31.272,-40.504,-179.918,5.424,148.923
C08007=1216.515,-31.522,-40.492,-179.921,5.424,148.923
C08008=1216.521,-31.771,-40.479,-179.923,5.424,148.924
C08009=1216.526,-32.021,-40.466,-179.926,5.424,148.925
C08010=1216.531,-32.271,-40.453,-179.928,5.423,148.925
C08011=1216.536,-32.520,-40.440,-179.930,5.423,148.926
C08012=1216.541,-32.770,-40.427,-179.933,5.423,148.927
C08013=1216.546,-33.020,-40.414,-179.936,5.422,148.928
C08014=1216.551,-33.269,-40.402,-179.938,5.423,148.928
C08015=1216.556,-33.519,-40.389,-179.940,5.422,148.929
C08016=1216.562,-33.769,-40.375,-179.943,5.422,148.930
C08017=1216.567,-34.018,-40.363,-179.945,5.422,148.930
C08018=1216.571,-34.268,-40.350,-179.947,5.421,148.931
C08019=1216.576,-34.517,-40.337,-179.950,5.421,148.931
C08020=1216.582,-34.767,-40.324,-179.952,5.421,148.932
C08021=1216.587,-35.017,-40.311,-179.955,5.421,148.933
C08022=1216.592,-35.266,-40.299,-179.957,5.420,148.934
C08023=1216.597,-35.516,-40.286,-179.960,5.420,148.934
C08024=1216.602,-35.765,-40.273,-179.962,5.420,148.935
C08025=1216.607,-36.015,-40.260,-179.965,5.419,148.936
C08026=1216.613,-36.264,-40.247,-179.967,5.420,148.936
C08027=1216.618,-36.514,-40.235,-179.970,5.419,148.937
C08028=1216.623,-36.763,-40.222,-179.972,5.419,148.938
C08029=1216.628,-37.014,-40.210,-179.974,5.419,148.938
C08030=1216.634,-37.263,-40.196,-179.977,5.419,148.939
C08031=1216.639,-37.513,-40.184,-179.980,5.418,148.940
C08032=1216.643,-37.763,-40.171,-179.982,5.419,148.941
C08033=1216.648,-38.012,-40.158,-179.984,5.418,148.941
C08034=1216.653,-38.261,-40.146,-179.987,5.418,148.942
C08035=1216.659,-38.511,-40.133,-179.989,5.418,148.943
C08036=1216.664,-38.761,-40.120,-179.992,5.417,148.943
C08037=1216.669,-39.011,-40.108,-179.994,5.418,148.944
C08038=1216.674,-39.260,-40.095,-179.996,5.417,148.945
C08039=1216.680,-39.510,-40.082,-179.999,5.416,148.945
C08040=1216.685,-39.759,-40.070,179.999,5.417,148.946
C08041=1216.689,-40.009,-40.057,179.997,5.416,148.947
C08042=1216.695,-40.259,-40.045,179.994,5.416,148.947
C08043=1216.700,-40.508,-40.032,179.992,5.416,148.948
C08044=1216.705,-40.757,-40.020,179.989,5.416,148.949
C08045=1216.709,-41.008,-40.007,179.986,5.415,148.949
C08046=1216.715,-41.257,-39.994,179.984,5.416,148.950
C08047=1216.721,-41.507,-39.982,179.982,5.415,148.951
C08048=1216.726,-41.756,-39.969,179.979,5.415,148.952
C08049=1216.731,-42.006,-39.957,179.977,5.415,148.952
C08050=1216.735,-42.256,-39.944,179.974,5.414,148.953
C08051=1216.741,-42.506,-39.932,179.972,5.414,148.954
C08052=1216.746,-42.755,-39.919,179.970,5.414,148.954
C08053=1216.751,-43.004,-39.907,179.967,5.414,148.955
C08054=1216.756,-43.254,-39.894,179.965,5.414,148.956
C08055=1216.761,-43.504,-39.882,179.962,5.414,148.956
C08056=1216.766,-43.754,-39.869,179.959,5.413,148.957
C08057=1216.771,-44.003,-39.856,179.957,5.414,148.958
C08058=1216.777,-44.253,-39.845,179.955,5.413,148.958
C08059=1216.782,-44.502,-39.832,179.953,5.412,148.959
C08060=1216.787,-44.751,-39.819,179.950,5.413,148.960
C08061=1216.792,-45.002,-39.807,179.948,5.412,148.960
C08062=1216.797,-45.251,-39.795,179.945,5.412,148.961
C08063=1216.802,-45.501,-39.782,179.943,5.412,148.962
C08064=1216.807,-45.751,-39.770,179.940,5.411,148.963
C08065=1216.813,-46.000,-39.757,179.938,5.412,148.963
C08066=1216.818,-46.249,-39.745,179.936,5.411,148.964
C08067=1216.823,-46.499,-39.733,179.933,5.411,148.965
C08068=1216.828,-46.749,-39.720,179.931,5.411,148.965
C08069=1216.833,-46.999,-39.708,179.928,5.411,148.966
C08070=1216.838,-47.249,-39.696,179.926,5.410,148.967
C08071=1216.843,-47.498,-39.683,179.923,5.411,148.967
C08072=1216.849,-47.748,-39.671,179.921,5.410,148.968
C08073=1216.854,-47.997,-39.658,179.919,5.410,148.969
C08074=1216.859,-48.247,-39.647,179.916,5.410,148.970
C08075=1216.864,-48.517,-39.633,179.913,5.410,148.970
C08076=1216.870,-48.787,-39.620,179.911,5.409,148.971
C08077=1216.876,-49.056,-39.606,179.909,5.409,148.972
C08078=1216.881,-49.327,-39.593,179.906,5.409,148.972
C08079=1216.886,-49.576,-39.580,179.903,5.408,148.973
C08080=1216.892,-49.826,-39.569,179.901,5.409,148.974
C08081=1216.896,-50.075,-39.557,179.899,5.408,148.974
C08082=1216.902,-50.325,-39.545,179.896,5.408,148.975
C08083=1216.907,-50.574,-39.532,179.894,5.408,148.976
C08084=1216.912,-50.824,-39.520,179.891,5.408,148.977
C08085=1216.917,-51.074,-39.508,179.889,5.408,148.977
C08086=1216.922,-51.324,-39.495,179.886,5.408,148.978
C08087=1216.927,-51.574,-39.483,179.884,5.407,148.979
C08088=1216.933,-51.823,-39.471,179.882,5.407,148.979
C08089=1216.937,-52.073,-39.460,179.879,5.407,148.980
C08090=1216.943,-52.322,-39.447,179.877,5.407,148.981
C08091=1216.948,-52.572,-39.435,179.874,5.407,148.982
C08092=1216.953,-52.822,-39.422,179.872,5.406,148.982
C08093=1216.959,-53.072,-39.411,179.870,5.406,148.983
C08094=1216.964,-53.321,-39.398,179.867,5.406,148.983
C08095=1216.968,-53.571,-39.387,179.865,5.406,148.984
C08096=1216.973,-53.820,-39.374,179.863,5.406,148.985
C08097=1216.979,-54.070,-39.362,179.860,5.405,148.986
C08098=1216.984,-54.320,-39.350,179.858,5.406,148.986
C08099=1216.989,-54.569,-39.338,179.855,5.405,148.987
C08100=1216.994,-54.819,-39.326,179.852,5.405,148.988
C08101=1217.000,-55.069,-39.315,179.850,5.405,148.988
C08102=1217.005,-55.318,-39.302,179.848,5.405,148.989
C08103=1217.010,-55.568,-39.290,179.846,5.405,148.990
C08104=1217.015,-55.817,-39.277,179.843,5.404,148.990
C08105=1217.020,-56.067,-39.266,179.840,5.404,148.991
C08106=1217.025,-56.317,-39.254,179.838,5.404,148.992
C08107=1217.030,-56.566,-39.242,179.836,5.404,148.993
C08108=1217.036,-56.816,-39.230,179.833,5.404,148.993
C08109=1217.041,-57.066,-39.218,179.831,5.404,148.994
C08110=1217.046,-57.315,-39.206,179.829,5.403,148.994
C08111=1217.051,-57.565,-39.194,179.827,5.403,148.995
C08112=1217.057,-57.815,-39.182,179.824,5.403,148.996
C08113=1217.061,-58.064,-39.171,179.822,5.403,148.997
C08114=1217.066,-58.314,-39.158,179.819,5.403,148.997
C08115=1217.072,-58.564,-39.146,179.817,5.403,148.998
C08116=1217.077,-58.813,-39.135,179.814,5.403,148.999
C08117=1217.082,-59.063,-39.123,179.812,5.402,148.999
C08118=1217.087,-59.313,-39.111,179.810,5.402,149.000
C08119=1217.093,-59.563,-39.099,179.807,5.402,149.001
C08120=1217.097,-59.812,-39.087,179.805,5.402,149.001
C08121=1217.103,-60.062,-39.075,179.802,5.402,149.002
C08122=1217.108,-60.311,-39.063,179.799,5.401,149.003
C08123=1217.112,-60.561,-39.052,179.797,5.402,149.004
C08124=1217.118,-60.811,-39.040,179.795,5.401,149.004
C08125=1217.123,-61.061,-39.028,179.793,5.401,149.005
C08126=1217.128,-61.310,-39.016,179.790,5.401,149.005
C08127=1217.133,-61.560,-39.004,179.788,5.400,149.006
C08128=1217.139,-61.810,-38.992,179.786,5.401,149.007
C08129=1217.143,-62.059,-38.981,179.783,5.400,149.008
C08130=1217.149,-62.309,-38.969,179.781,5.401,149.008
C08131=1217.155,-62.559,-38.957,179.778,5.400,149.009
C08132=1217.159,-62.808,-38.945,179.776,5.400,149.010
C08133=1217.165,-63.058,-38.933,179.774,5.400,149.010
C08134=1217.169,-63.307,-38.922,179.771,5.400,149.011
C08135=1217.175,-63.557,-38.910,179.769,5.400,149.012
C08136=1217.180,-63.807,-38.898,179.766,5.399,149.013
C08137=1217.185,-64.057,-38.887,179.764,5.400,149.013
C08138=1217.190,-64.307,-38.875,179.761,5.399,149.014
C08139=1217.196,-64.557,-38.863,179.759,5.399,149.014
C08140=1217.200,-64.806,-38.852,179.757,5.399,149.015
C08141=1217.206,-65.055,-38.840,179.754,5.398,149.016
C08142=1217.211,-65.304,-38.829,179.752,5.399,149.017
C08143=1217.216,-65.554,-38.817,179.750,5.398,149.017
C08144=1217.221,-65.804,-38.805,179.748,5.399,149.018
C08145=1217.226,-66.054,-38.793,179.745,5.398,149.019
C08146=1217.232,-66.304,-38.782,179.742,5.398,149.019
C08147=1217.236,-66.553,-38.770,179.740,5.398,149.020
C08148=1217.242,-66.803,-38.758,179.737,5.398,149.021
C08149=1217.247,-67.052,-38.747,179.735,5.398,149.022
C08150=1217.253,-67.302,-38.736,179.733,5.398,149.022
C08151=1217.257,-67.552,-38.724,179.731,5.398,149.023
C08152=1217.263,-67.802,-38.712,179.728,5.397,149.024
C08153=1217.267,-68.051,-38.701,179.726,5.397,149.024
C08154=1217.273,-68.301,-38.689,179.724,5.397,149.025
C08155=1217.278,-68.550,-38.678,179.721,5.396,149.026
C08156=1217.284,-68.800,-38.666,179.719,5.397,149.026
C08157=1217.288,-69.050,-38.655,179.716,5.396,149.027
C08158=1217.294,-69.300,-38.643,179.714,5.397,149.028
C08159=1217.298,-69.549,-38.632,179.712,5.396,149.028
C08160=1217.304,-69.799,-38.620,179.709,5.397,149.029
C08161=1217.309,-70.048,-38.609,179.707,5.396,149.030
C08162=1217.314,-70.298,-38.597,179.704,5.396,149.030
C08163=1217.319,-70.548,-38.586,179.702,5.396,149.031
C08164=1217.325,-70.798,-38.574,179.699,5.396,149.032
C08165=1217.330,-71.048,-38.564,179.698,5.396,149.032
C08166=1217.336,-71.297,-38.552,179.695,5.395,149.033
C08167=1217.340,-71.547,-38.541,179.693,5.395,149.034
C08168=1217.346,-71.797,-38.529,179.690,5.395,149.034
C08169=1217.350,-72.046,-38.518,179.688,5.395,149.035
C08170=1217.356,-72.296,-38.506,179.686,5.395,149.036
C08171=1217.361,-72.545,-38.495,179.683,5.394,149.037
C08172=1217.367,-72.795,-38.483,179.681,5.395,149.037
C08173=1217.371,-73.045,-38.472,179.678,5.394,149.038
C08174=1217.376,-73.295,-38.461,179.676,5.395,149.039
C08175=1217.382,-73.544,-38.449,179.673,5.394,149.039
C08176=1217.387,-73.794,-38.438,179.671,5.395,149.040
C08177=1217.392,-74.044,-38.426,179.669,5.394,149.041
C08178=1217.397,-74.294,-38.415,179.667,5.394,149.041
C08179=1217.403,-74.564,-38.403,179.664,5.394,149.042
C08180=1217.409,-74.835,-38.391,179.661,5.394,149.043
C08181=1217.414,-75.105,-38.378,179.659,5.393,149.044
C08182=1217.420,-75.375,-38.366,179.656,5.394,149.044
C08183=1217.425,-75.625,-38.355,179.654,5.393,149.045
C08184=1217.430,-75.875,-38.344,179.652,5.393,149.046
C08185=1217.436,-76.125,-38.333,179.649,5.393,149.047
C08186=1217.441,-76.374,-38.321,179.647,5.393,149.047
C08187=1217.446,-76.624,-38.310,179.644,5.393,149.048
C08188=1217.452,-76.874,-38.299,179.643,5.393,149.048
C08189=1217.457,-77.123,-38.288,179.640,5.392,149.049
C08190=1217.461,-77.373,-38.277,179.637,5.392,149.050
C08191=1217.467,-77.623,-38.265,179.635,5.392,149.051
C08192=1217.472,-77.872,-38.255,179.633,5.392,149.051
C08193=1217.477,-78.122,-38.243,179.630,5.392,149.052
C08194=1217.482,-78.372,-38.231,179.628,5.392,149.053
C08195=1217.488,-78.621,-38.220,179.626,5.392,149.053
C08196=1217.493,-78.871,-38.210,179.623,5.392,149.054
C08197=1217.498,-79.121,-38.198,179.621,5.392,149.055
C08198=1217.503,-79.371,-38.187,179.619,5.391,149.055
C08199=1217.508,-79.620,-38.177,179.617,5.392,149.056
C08200=1217.514,-79.870,-38.165,179.614,5.391,149.057
C08201=1217.519,-80.120,-38.153,179.611,5.391,149.057
C08202=1217.524,-80.369,-38.143,179.609,5.391,149.058
C08203=1217.529,-80.619,-38.132,179.607,5.391,149.059
C08204=1217.534,-80.869,-38.120,179.604,5.391,149.060
C08205=1217.540,-81.118,-38.110,179.602,5.391,149.060
C08206=1217.545,-81.368,-38.098,179.600,5.391,149.061
C08207=1217.550,-81.619,-38.087,179.597,5.391,149.062
C08208=1217.556,-81.868,-38.076,179.595,5.390,149.062
C08209=1217.560,-82.117,-38.065,179.593,5.390,149.063
C08210=1217.565,-82.367,-38.055,179.591,5.390,149.064
C08211=1217.571,-82.616,-38.044,179.588,5.390,149.064
C08212=1217.576,-82.867,-38.032,179.586,5.390,149.065
C08213=1217.582,-83.116,-38.021,179.583,5.390,149.066
C08214=1217.586,-83.365,-38.010,179.581,5.390,149.066
C08215=1217.591,-83.616,-38.000,179.578,5.390,149.067
C08216=1217.597,-83.865,-37.988,179.576,5.389,149.068
C08217=1217.602,-84.115,-37.978,179.574,5.390,149.069
C08218=1217.607,-84.365,-37.966,179.572,5.389,149.069
C08219=1217.613,-84.614,-37.956,179.569,5.389,149.070
C08220=1217.617,-84.864,-37.945,179.567,5.389,149.070
C08221=1217.623,-85.114,-37.934,179.565,5.389,149.071
C08222=1217.628,-85.363,-37.923,179.562,5.389,149.072
C08223=1217.633,-85.614,-37.912,179.560,5.389,149.073
C08224=1217.639,-85.863,-37.901,179.557,5.389,149.073
C08225=1217.644,-86.113,-37.891,179.555,5.389,149.074
C08226=1217.648,-86.362,-37.879,179.552,5.389,149.075
C08227=1217.654,-86.612,-37.869,179.551,5.389,149.075
C08228=1217.659,-86.862,-37.857,179.548,5.388,149.076
C08229=1217.665,-87.111,-37.847,179.546,5.388,149.077
C08230=1217.670,-87.361,-37.836,179.543,5.388,149.077
C08231=1217.675,-87.611,-37.825,179.541,5.388,149.078
C08232=1217.680,-87.860,-37.814,179.539,5.388,149.079
C08233=1217.685,-88.111,-37.804,179.537,5.388,149.079
C08234=1217.690,-88.359,-37.793,179.534,5.388,149.080
C08235=1217.696,-88.610,-37.782,179.532,5.388,149.081
C08236=1217.701,-88.859,-37.771,179.530,5.387,149.081
C08237=1217.706,-89.109,-37.760,179.528,5.388,149.082
C08238=1217.712,-89.359,-37.750,179.525,5.387,149.083
C08239=1217.717,-89.608,-37.739,179.522,5.387,149.083
C08240=1217.722,-89.859,-37.728,179.520,5.387,149.084
C08241=1217.727,-90.107,-37.717,179.517,5.387,149.085
C08242=1217.732,-90.358,-37.706,179.515,5.387,149.086
C08243=1217.737,-90.607,-37.696,179.513,5.387,149.086
C08244=1217.742,-90.857,-37.685,179.511,5.387,149.087
C08245=1217.748,-91.106,-37.675,179.508,5.386,149.088
C08246=1217.753,-91.357,-37.664,179.506,5.387,149.088
C08247=1217.759,-91.606,-37.653,179.504,5.386,149.089
C08248=1217.764,-91.856,-37.642,179.502,5.387,149.090
C08249=1217.769,-92.106,-37.632,179.499,5.386,149.090
C08250=1217.774,-92.355,-37.621,179.497,5.387,149.091
C08251=1217.780,-92.605,-37.610,179.495,5.386,149.092
C08252=1217.785,-92.855,-37.600,179.493,5.386,149.092
C08253=1217.790,-93.104,-37.589,179.490,5.386,149.093
C08254=1217.795,-93.354,-37.578,179.488,5.386,149.094
C08255=1217.801,-93.604,-37.568,179.485,5.386,149.094
C08256=1217.806,-93.854,-37.558,179.483,5.386,149.095
C08257=1217.811,-94.103,-37.547,179.480,5.386,149.096
C08258=1217.816,-94.353,-37.536,179.478,5.386,149.097
C08259=1217.821,-94.603,-37.526,179.476,5.385,149.097
C08260=1217.826,-94.852,-37.515,179.474,5.385,149.098
C08261=1217.832,-95.102,-37.504,179.471,5.385,149.098
C08262=1217.837,-95.352,-37.494,179.469,5.385,149.099
C08263=1217.842,-95.602,-37.484,179.467,5.385,149.100
C08264=1217.847,-95.852,-37.473,179.464,5.385,149.101
C08265=1217.853,-96.101,-37.462,179.462,5.385,149.101
C08266=1217.858,-96.351,-37.451,179.460,5.385,149.102
C08267=1217.863,-96.601,-37.441,179.457,5.384,149.102
C08268=1217.868,-96.851,-37.431,179.455,5.385,149.103
C08269=1217.873,-97.100,-37.420,179.453,5.384,149.104
C08270=1217.879,-97.349,-37.410,179.451,5.385,149.105
C08271=1217.884,-97.600,-37.399,179.448,5.384,149.105
C08272=1217.889,-97.849,-37.389,179.446,5.385,149.106
C08273=1217.894,-98.099,-37.379,179.444,5.384,149.107
C08274=1217.900,-98.349,-37.369,179.442,5.384,149.107
C08275=1217.904,-98.598,-37.357,179.439,5.384,149.108
C08276=1217.910,-98.848,-37.347,179.437,5.384,149.109
C08277=1217.915,-99.098,-37.336,179.434,5.384,149.109
C08278=1217.920,-99.348,-37.326,179.432,5.384,149.110
C08279=1217.926,-99.597,-37.316,179.429,5.384,149.111
C08280=1217.931,-99.847,-37.305,179.428,5.384,149.111
C08281=1217.937,-100.097,-37.295,179.425,5.383,149.112
C08282=1217.942,-100.347,-37.285,179.423,5.384,149.113
C08283=1217.947,-100.617,-37.273,179.420,5.383,149.113
C08284=1217.952,-100.888,-37.262,179.418,5.384,149.114
C08285=1217.958,-101.160,-37.251,179.416,5.383,149.115
C08286=1217.964,-101.431,-37.240,179.413,5.383,149.116
C08287=1217.969,-101.681,-37.230,179.411,5.383,149.116
C08288=1217.975,-101.930,-37.220,179.408,5.383,149.117
C08289=1217.980,-102.181,-37.209,179.406,5.383,149.118
C08290=1217.985,-102.430,-37.199,179.403,5.383,149.118
C08291=1217.991,-102.680,-37.189,179.401,5.383,149.119
C08292=1217.995,-102.930,-37.179,179.399,5.383,149.120
C08293=1218.001,-103.179,-37.168,179.397,5.383,149.120
C08294=1218.006,-103.430,-37.158,179.394,5.382,149.121
C08295=1218.011,-103.679,-37.148,179.392,5.383,149.122
C08296=1218.017,-103.929,-37.137,179.390,5.382,149.122
C08297=1218.022,-104.178,-37.126,179.387,5.382,149.123
C08298=1218.026,-104.427,-37.117,179.385,5.382,149.124
C08299=1218.032,-104.678,-37.107,179.383,5.382,149.124
C08300=1218.037,-104.928,-37.096,179.381,5.382,149.125
C08301=1218.043,-105.177,-37.086,179.378,5.382,149.126
C08302=1218.048,-105.427,-37.076,179.376,5.382,149.127
C08303=1218.053,-105.677,-37.066,179.374,5.382,149.127
C08304=1218.058,-105.926,-37.056,179.372,5.382,149.128
C08305=1218.064,-106.176,-37.046,179.369,5.382,149.128
C08306=1218.069,-106.426,-37.035,179.367,5.382,149.129
C08307=1218.074,-106.675,-37.025,179.365,5.381,149.130
C08308=1218.079,-106.925,-37.015,179.363,5.382,149.131
C08309=1218.084,-107.175,-37.005,179.360,5.381,149.131
C08310=1218.090,-107.425,-36.994,179.358,5.382,149.132
C08311=1218.095,-107.674,-36.985,179.356,5.381,149.133
C08312=1218.100,-107.924,-36.974,179.353,5.381,149.133
C08313=1218.105,-108.174,-36.964,179.351,5.381,149.134
C08314=1218.111,-108.423,-36.954,179.349,5.381,149.135
C08315=1218.116,-108.674,-36.945,179.346,5.381,149.135
C08316=1218.121,-108.923,-36.934,179.344,5.381,149.136
C08317=1218.127,-109.173,-36.924,179.342,5.380,149.137
C08318=1218.131,-109.423,-36.914,179.340,5.381,149.137
C08319=1218.137,-109.672,-36.904,179.337,5.380,149.138
C08320=1218.142,-109.922,-36.894,179.335,5.381,149.139
C08321=1218.148,-110.172,-36.884,179.332,5.380,149.139
C08322=1218.152,-110.422,-36.874,179.331,5.380,149.140
C08323=1218.158,-110.672,-36.864,179.328,5.380,149.141
C08324=1218.164,-110.921,-36.854,179.326,5.380,149.141
C08325=1218.168,-111.170,-36.844,179.324,5.381,149.142
C08326=1218.173,-111.421,-36.834,179.321,5.380,149.143
C08327=1218.179,-111.670,-36.823,179.319,5.380,149.143
C08328=1218.184,-111.920,-36.815,179.317,5.380,149.144
C08329=1218.190,-112.170,-36.804,179.315,5.380,149.145
C08330=1218.195,-112.420,-36.794,179.312,5.380,149.145
C08331=1218.200,-112.669,-36.784,179.310,5.380,149.146
C08332=1218.206,-112.919,-36.775,179.308,5.379,149.147
C08333=1218.211,-113.169,-36.764,179.306,5.380,149.147
C08334=1218.215,-113.419,-36.755,179.303,5.379,149.148
C08335=1218.221,-113.668,-36.744,179.301,5.380,149.149
C08336=1218.226,-113.918,-36.735,179.298,5.379,149.149
C08337=1218.232,-114.168,-36.725,179.297,5.379,149.150
C08338=1218.237,-114.418,-36.715,179.294,5.379,149.151
C08339=1218.242,-114.667,-36.705,179.292,5.379,149.151
C08340=1218.248,-114.917,-36.696,179.289,5.379,149.152
C08341=1218.253,-115.167,-36.685,179.287,5.379,149.153
C08342=1218.258,-115.416,-36.676,179.285,5.379,149.153
C08343=1218.263,-115.667,-36.666,179.283,5.379,149.154
C08344=1218.268,-115.916,-36.656,179.281,5.379,149.155
C08345=1218.274,-116.166,-36.646,179.278,5.379,149.155
C08346=1218.279,-116.416,-36.637,179.276,5.379,149.156
C08347=1218.285,-116.665,-36.627,179.274,5.378,149.157
C08348=1218.290,-116.915,-36.616,179.272,5.379,149.157
C08349=1218.295,-117.165,-36.607,179.269,5.378,149.158
C08350=1218.300,-117.415,-36.597,179.267,5.379,149.159
C08351=1218.305,-117.664,-36.588,179.264,5.378,149.160
C08352=1218.311,-117.914,-36.578,179.263,5.378,149.160
C08353=1218.315,-118.164,-36.568,179.260,5.378,149.161
C08354=1218.321,-118.414,-36.558,179.258,5.378,149.161
C08355=1218.326,-118.663,-36.549,179.255,5.378,149.162
C08356=1218.332,-118.913,-36.539,179.254,5.378,149.163
C08357=1218.337,-119.162,-36.529,179.251,5.378,149.163
C08358=1218.342,-119.412,-36.520,179.249,5.378,149.164
C08359=1218.347,-119.662,-36.510,179.247,5.378,149.165
C08360=1218.353,-119.913,-36.500,179.244,5.378,149.165
C08361=1218.358,-120.162,-36.491,179.242,5.378,149.166
C08362=1218.363,-120.412,-36.481,179.240,5.377,149.167
C08363=1218.368,-120.661,-36.472,179.238,5.378,149.167
C08364=1218.374,-120.911,-36.461,179.235,5.377,149.168
C08365=1218.378,-121.161,-36.452,179.233,5.377,149.169
C08366=1218.384,-121.411,-36.442,179.231,5.377,149.169
C08367=1218.389,-121.661,-36.433,179.229,5.377,149.170
C08368=1218.395,-121.910,-36.423,179.226,5.378,149.171
C08369=1218.400,-122.160,-36.414,179.224,5.377,149.171
C08370=1218.406,-122.410,-36.404,179.222,5.377,149.172
C08371=1218.411,-122.659,-36.395,179.220,5.377,149.173
C08372=1218.416,-122.909,-36.385,179.217,5.377,149.173
C08373=1218.421,-123.160,-36.375,179.215,5.377,149.174
C08374=1218.427,-123.409,-36.365,179.213,5.377,149.175
C08375=1218.432,-123.659,-36.356,179.210,5.376,149.175
C08376=1218.437,-123.908,-36.347,179.208,5.377,149.176
C08377=1218.442,-124.158,-36.337,179.206,5.376,149.177
C08378=1218.447,-124.408,-36.327,179.204,5.376,149.177
C08379=1218.453,-124.658,-36.318,179.202,5.377,149.178
C08380=1218.458,-124.907,-36.308,179.199,5.376,149.179
C08381=1218.463,-125.157,-36.299,179.197,5.377,149.179
C08382=1218.469,-125.406,-36.289,179.195,5.376,149.180
C08383=1218.473,-125.657,-36.280,179.193,5.376,149.181
C08384=1218.479,-125.907,-36.270,179.190,5.376,149.181
C08385=1218.484,-126.156,-36.261,179.188,5.376,149.182
C08386=1218.489,-126.406,-36.252,179.186,5.376,149.183
C08387=1218.068,-126.416,-36.289,179.182,5.379,149.185
C08388=1218.063,-126.167,-36.298,179.184,5.380,149.184
C08389=1218.058,-125.917,-36.307,179.186,5.379,149.183
C08390=1218.052,-125.667,-36.317,179.189,5.380,149.183
C08391=1218.047,-125.418,-36.326,179.191,5.380,149.182
C08392=1218.041,-125.168,-36.336,179.193,5.380,149.181
C08393=1218.037,-124.918,-36.345,179.195,5.380,149.181
C08394=1218.031,-124.668,-36.354,179.198,5.380,149.180
C08395=1218.026,-124.419,-36.364,179.200,5.380,149.179
C08396=1218.021,-124.169,-36.373,179.202,5.380,149.179
C08397=1218.015,-123.920,-36.384,179.204,5.380,149.178
C08398=1218.010,-123.670,-36.392,179.206,5.380,149.177
C08399=1218.005,-123.419,-36.403,179.209,5.380,149.177
C08400=1218.000,-123.170,-36.412,179.211,5.380,149.176
C08401=1217.995,-122.920,-36.421,179.213,5.380,149.175
C08402=1217.989,-122.670,-36.431,179.215,5.380,149.175
C08403=1217.984,-122.420,-36.440,179.218,5.381,149.174
C08404=1217.978,-122.171,-36.450,179.220,5.380,149.173
C08405=1217.973,-121.922,-36.460,179.223,5.381,149.173
C08406=1217.967,-121.671,-36.469,179.224,5.381,149.172
C08407=1217.963,-121.421,-36.479,179.226,5.381,149.171
C08408=1217.957,-121.171,-36.489,179.229,5.381,149.171
C08409=1217.952,-120.922,-36.498,179.231,5.381,149.170
C08410=1217.947,-120.672,-36.508,179.234,5.381,149.169
C08411=1217.942,-120.423,-36.517,179.235,5.381,149.169
C08412=1217.936,-120.172,-36.527,179.238,5.381,149.168
C08413=1217.931,-119.923,-36.537,179.240,5.381,149.167
C08414=1217.926,-119.672,-36.546,179.243,5.381,149.167
C08415=1217.921,-119.423,-36.556,179.244,5.381,149.166
C08416=1217.915,-119.174,-36.566,179.247,5.382,149.165
C08417=1217.910,-118.924,-36.575,179.249,5.381,149.165
C08418=1217.904,-118.674,-36.585,179.251,5.381,149.164
C08419=1217.899,-118.424,-36.594,179.254,5.381,149.163
C08420=1217.894,-118.174,-36.605,179.255,5.381,149.163
C08421=1217.889,-117.925,-36.614,179.258,5.382,149.162
C08422=1217.883,-117.675,-36.624,179.260,5.381,149.161
C08423=1217.879,-117.426,-36.634,179.263,5.382,149.161
C08424=1217.873,-117.176,-36.644,179.265,5.382,149.160
C08425=1217.868,-116.926,-36.653,179.267,5.382,149.159
C08426=1217.863,-116.676,-36.663,179.269,5.382,149.159
C08427=1217.858,-116.427,-36.673,179.272,5.382,149.158
C08428=1217.852,-116.176,-36.682,179.274,5.382,149.157
C08429=1217.846,-115.927,-36.693,179.276,5.383,149.157
C08430=1217.842,-115.678,-36.702,179.278,5.382,149.156
C08431=1217.836,-115.427,-36.712,179.281,5.383,149.155
C08432=1217.831,-115.178,-36.722,179.283,5.382,149.155
C08433=1217.826,-114.928,-36.732,179.285,5.382,149.154
C08434=1217.820,-114.678,-36.741,179.287,5.383,149.153
C08435=1217.815,-114.429,-36.751,179.289,5.382,149.153
C08436=1217.810,-114.178,-36.762,179.292,5.383,149.152
C08437=1217.805,-113.929,-36.771,179.294,5.382,149.151
C08438=1217.799,-113.679,-36.781,179.297,5.383,149.151
C08439=1217.794,-113.429,-36.791,179.299,5.383,149.150
C08440=1217.789,-113.180,-36.801,179.301,5.383,149.149
C08441=1217.784,-112.930,-36.811,179.303,5.383,149.149
C08442=1217.778,-112.680,-36.821,179.306,5.383,149.148
C08443=1217.773,-112.431,-36.830,179.308,5.383,149.147
C08444=1217.768,-112.180,-36.841,179.310,5.384,149.147
C08445=1217.762,-111.931,-36.851,179.312,5.383,149.146
C08446=1217.757,-111.681,-36.860,179.315,5.384,149.145
C08447=1217.752,-111.431,-36.870,179.317,5.383,149.145
C08448=1217.747,-111.181,-36.881,179.320,5.384,149.144
C08449=1217.742,-110.932,-36.890,179.321,5.384,149.143
C08450=1217.736,-110.682,-36.900,179.323,5.384,149.143
C08451=1217.731,-110.433,-36.911,179.326,5.384,149.142
C08452=1217.726,-110.182,-36.920,179.328,5.384,149.141
C08453=1217.721,-109.933,-36.930,179.331,5.384,149.141
C08454=1217.715,-109.683,-36.940,179.333,5.384,149.140
C08455=1217.711,-109.433,-36.950,179.335,5.384,149.139
C08456=1217.705,-109.184,-36.961,179.337,5.384,149.139
C08457=1217.699,-108.934,-36.971,179.340,5.384,149.138
C08458=1217.694,-108.684,-36.980,179.342,5.384,149.137
C08459=1217.689,-108.434,-36.990,179.344,5.385,149.137
C08460=1217.684,-108.185,-37.000,179.346,5.384,149.136
C08461=1217.678,-107.935,-37.011,179.349,5.385,149.135
C08462=1217.674,-107.685,-37.021,179.351,5.385,149.135
C08463=1217.668,-107.436,-37.031,179.354,5.385,149.134
C08464=1217.663,-107.186,-37.041,179.356,5.385,149.133
C08465=1217.658,-106.936,-37.052,179.358,5.385,149.133
C08466=1217.653,-106.687,-37.061,179.360,5.385,149.132
C08467=1217.647,-106.437,-37.071,179.363,5.385,149.131
C08468=1217.642,-106.187,-37.082,179.365,5.385,149.131
C08469=1217.636,-105.937,-37.091,179.368,5.385,149.130
C08470=1217.631,-105.687,-37.101,179.370,5.385,149.129
C08471=1217.626,-105.437,-37.112,179.372,5.386,149.129
C08472=1217.621,-105.188,-37.122,179.374,5.386,149.128
C08473=1217.615,-104.938,-37.132,179.377,5.386,149.127
C08474=1217.610,-104.688,-37.143,179.379,5.386,149.127
C08475=1217.605,-104.439,-37.152,179.381,5.385,149.126
C08476=1217.600,-104.189,-37.162,179.384,5.386,149.125
C08477=1217.595,-103.939,-37.173,179.385,5.386,149.125
C08478=1217.589,-103.689,-37.183,179.388,5.386,149.124
C08479=1217.584,-103.440,-37.193,179.390,5.386,149.123
C08480=1217.579,-103.190,-37.203,179.393,5.386,149.122
C08481=1217.574,-102.940,-37.214,179.395,5.386,149.122
C08482=1217.569,-102.690,-37.224,179.397,5.386,149.121
C08483=1217.563,-102.440,-37.234,179.399,5.386,149.121
C08484=1217.558,-102.191,-37.245,179.402,5.387,149.120
C08485=1217.553,-101.941,-37.256,179.404,5.386,149.119
C08486=1217.548,-101.692,-37.266,179.406,5.387,149.118
C08487=1217.542,-101.442,-37.276,179.408,5.386,149.118
C08488=1217.536,-101.171,-37.287,179.411,5.387,149.117
C08489=1217.531,-100.900,-37.298,179.414,5.387,149.116
C08490=1217.525,-100.628,-37.310,179.416,5.387,149.116
C08491=1217.520,-100.357,-37.320,179.419,5.387,149.115
C08492=1217.515,-100.107,-37.331,179.421,5.387,149.114
C08493=1217.509,-99.858,-37.341,179.423,5.387,149.113
C08494=1217.504,-99.608,-37.352,179.425,5.387,149.113
C08495=1217.499,-99.358,-37.363,179.428,5.388,149.112
C08496=1217.493,-99.109,-37.373,179.430,5.387,149.111
C08497=1217.489,-98.859,-37.383,179.432,5.388,149.111
C08498=1217.483,-98.609,-37.393,179.434,5.387,149.110
C08499=1217.478,-98.359,-37.404,179.437,5.388,149.109
C08500=1217.473,-98.110,-37.414,179.439,5.387,149.109
C08501=1217.468,-97.860,-37.425,179.442,5.388,149.108
C08502=1217.462,-97.610,-37.435,179.444,5.388,149.107
C08503=1217.457,-97.361,-37.446,179.446,5.388,149.107
C08504=1217.452,-97.111,-37.456,179.448,5.388,149.106
C08505=1217.446,-96.861,-37.466,179.451,5.388,149.105
C08506=1217.441,-96.611,-37.477,179.453,5.388,149.105
C08507=1217.436,-96.362,-37.488,179.456,5.388,149.104
C08508=1217.431,-96.112,-37.498,179.458,5.388,149.103
C08509=1217.425,-95.862,-37.509,179.460,5.389,149.103
C08510=1217.420,-95.612,-37.519,179.462,5.388,149.102
C08511=1217.415,-95.363,-37.530,179.465,5.389,149.101
C08512=1217.410,-95.113,-37.541,179.467,5.389,149.101
C08513=1217.404,-94.863,-37.551,179.470,5.389,149.100
C08514=1217.399,-94.614,-37.561,179.472,5.389,149.099
C08515=1217.394,-94.363,-37.572,179.474,5.389,149.098
C08516=1217.388,-94.114,-37.583,179.476,5.389,149.098
C08517=1217.383,-93.864,-37.593,179.479,5.389,149.097
C08518=1217.378,-93.615,-37.603,179.481,5.389,149.097
C08519=1217.373,-93.365,-37.615,179.483,5.390,149.096
C08520=1217.368,-93.116,-37.625,179.485,5.389,149.095
C08521=1217.363,-92.865,-37.635,179.488,5.390,149.094
C08522=1217.357,-92.616,-37.646,179.490,5.389,149.094
C08523=1217.352,-92.366,-37.657,179.492,5.390,149.093
C08524=1217.347,-92.117,-37.667,179.494,5.390,149.092
C08525=1217.342,-91.866,-37.678,179.497,5.390,149.092
C08526=1217.336,-91.617,-37.689,179.499,5.390,149.091
C08527=1217.331,-91.367,-37.699,179.502,5.390,149.090
C08528=1217.326,-91.117,-37.710,179.504,5.390,149.090
C08529=1217.321,-90.868,-37.721,179.507,5.390,149.089
C08530=1217.316,-90.618,-37.731,179.509,5.390,149.088
C08531=1217.311,-90.369,-37.742,179.511,5.391,149.088
C08532=1217.306,-90.119,-37.753,179.514,5.391,149.087
C08533=1217.300,-89.869,-37.763,179.516,5.391,149.086
C08534=1217.295,-89.619,-37.775,179.518,5.391,149.086
C08535=1217.289,-89.370,-37.785,179.520,5.391,149.085
C08536=1217.284,-89.119,-37.796,179.523,5.391,149.084
C08537=1217.279,-88.870,-37.807,179.525,5.391,149.083
C08538=1217.274,-88.620,-37.817,179.528,5.391,149.083
C08539=1217.269,-88.370,-37.828,179.529,5.391,149.082
C08540=1217.264,-88.121,-37.839,179.532,5.392,149.082
C08541=1217.259,-87.871,-37.850,179.534,5.391,149.081
C08542=1217.253,-87.622,-37.860,179.537,5.392,149.080
C08543=1217.248,-87.372,-37.871,179.539,5.392,149.079
C08544=1217.242,-87.122,-37.882,179.542,5.392,149.079
C08545=1217.237,-86.872,-37.893,179.544,5.392,149.078
C08546=1217.233,-86.622,-37.904,179.546,5.392,149.077
C08547=1217.227,-86.373,-37.914,179.548,5.392,149.077
C08548=1217.222,-86.123,-37.926,179.551,5.393,149.076
C08549=1217.217,-85.874,-37.936,179.553,5.392,149.075
C08550=1217.211,-85.624,-37.948,179.555,5.393,149.075
C08551=1217.206,-85.374,-37.958,179.558,5.392,149.074
C08552=1217.201,-85.125,-37.969,179.560,5.393,149.073
C08553=1217.196,-84.874,-37.980,179.562,5.392,149.073
C08554=1217.191,-84.625,-37.991,179.565,5.393,149.072
C08555=1217.186,-84.375,-38.001,179.568,5.393,149.071
C08556=1217.180,-84.125,-38.013,179.569,5.393,149.071
C08557=1217.175,-83.876,-38.023,179.572,5.394,149.070
C08558=1217.170,-83.626,-38.035,179.574,5.393,149.069
C08559=1217.165,-83.376,-38.046,179.577,5.394,149.069
C08560=1217.160,-83.127,-38.056,179.579,5.393,149.068
C08561=1217.154,-82.877,-38.068,179.581,5.394,149.067
C08562=1217.149,-82.627,-38.078,179.584,5.393,149.066
C08563=1217.144,-82.378,-38.090,179.586,5.394,149.066
C08564=1217.139,-82.128,-38.100,179.588,5.394,149.065
C08565=1217.133,-81.878,-38.112,179.591,5.394,149.064
C08566=1217.128,-81.629,-38.123,179.593,5.394,149.064
C08567=1217.123,-81.378,-38.134,179.595,5.394,149.063
C08568=1217.118,-81.130,-38.144,179.597,5.394,149.062
C08569=1217.113,-80.880,-38.156,179.600,5.395,149.062
C08570=1217.108,-80.629,-38.167,179.603,5.395,149.061
C08571=1217.102,-80.380,-38.178,179.605,5.395,149.060
C08572=1217.097,-80.130,-38.188,179.607,5.395,149.060
C08573=1217.092,-79.880,-38.200,179.610,5.395,149.059
C08574=1217.087,-79.631,-38.211,179.612,5.395,149.058
C08575=1217.082,-79.381,-38.222,179.614,5.395,149.058
C08576=1217.076,-79.131,-38.234,179.616,5.396,149.057
C08577=1217.071,-78.882,-38.245,179.619,5.395,149.056
C08578=1217.066,-78.633,-38.256,179.621,5.396,149.055
C08579=1217.061,-78.382,-38.266,179.623,5.395,149.055
C08580=1217.056,-78.132,-38.278,179.626,5.396,149.054
C08581=1217.050,-77.883,-38.289,179.628,5.395,149.053
C08582=1217.045,-77.633,-38.300,179.631,5.396,149.053
C08583=1217.040,-77.383,-38.312,179.633,5.396,149.052
C08584=1217.035,-77.134,-38.323,179.636,5.396,149.051
C08585=1217.030,-76.885,-38.334,179.638,5.397,149.051
C08586=1217.024,-76.634,-38.345,179.640,5.396,149.050
C08587=1217.020,-76.385,-38.356,179.642,5.397,149.049
C08588=1217.014,-76.135,-38.368,179.645,5.397,149.049
C08589=1217.009,-75.886,-38.379,179.647,5.397,149.048
C08590=1217.004,-75.635,-38.390,179.649,5.397,149.047
C08591=1216.998,-75.386,-38.401,179.652,5.397,149.047
C08592=1216.993,-75.116,-38.413,179.655,5.397,149.046
C08593=1216.988,-74.845,-38.426,179.657,5.397,149.045
C08594=1216.981,-74.575,-38.438,179.659,5.398,149.044
C08595=1216.976,-74.304,-38.450,179.662,5.398,149.044
C08596=1216.971,-74.054,-38.461,179.664,5.398,149.043
C08597=1216.965,-73.805,-38.473,179.667,5.398,149.042
C08598=1216.960,-73.555,-38.484,179.669,5.398,149.042
C08599=1216.955,-73.306,-38.496,179.672,5.398,149.041
C08600=1216.950,-73.055,-38.507,179.674,5.398,149.040
C08601=1216.945,-72.805,-38.518,179.676,5.398,149.039
C08602=1216.939,-72.556,-38.529,179.679,5.399,149.039
C08603=1216.935,-72.307,-38.541,179.681,5.398,149.038
C08604=1216.929,-72.057,-38.553,179.684,5.399,149.037
C08605=1216.924,-71.807,-38.564,179.686,5.399,149.037
C08606=1216.918,-71.558,-38.575,179.688,5.399,149.036
C08607=1216.913,-71.308,-38.586,179.690,5.399,149.035
C08608=1216.908,-71.058,-38.598,179.693,5.399,149.035
C08609=1216.903,-70.808,-38.609,179.695,5.399,149.034
C08610=1216.898,-70.558,-38.621,179.698,5.400,149.033
C08611=1216.893,-70.309,-38.632,179.700,5.400,149.033
C08612=1216.887,-70.059,-38.644,179.702,5.400,149.032
C08613=1216.882,-69.810,-38.655,179.705,5.400,149.031
C08614=1216.877,-69.560,-38.667,179.707,5.400,149.030
C08615=1216.872,-69.310,-38.678,179.710,5.400,149.030
C08616=1216.866,-69.061,-38.690,179.712,5.400,149.029
C08617=1216.862,-68.811,-38.701,179.715,5.400,149.028
C08618=1216.856,-68.561,-38.713,179.716,5.400,149.028
C08619=1216.851,-68.312,-38.724,179.719,5.401,149.027
C08620=1216.846,-68.062,-38.736,179.721,5.401,149.026
C08621=1216.841,-67.812,-38.747,179.724,5.401,149.026
C08622=1216.835,-67.563,-38.759,179.726,5.401,149.025
C08623=1216.831,-67.313,-38.770,179.728,5.401,149.024
C08624=1216.825,-67.063,-38.782,179.731,5.401,149.024
C08625=1216.821,-66.814,-38.793,179.733,5.401,149.023
C08626=1216.815,-66.564,-38.805,179.736,5.402,149.022
C08627=1216.810,-66.314,-38.817,179.738,5.402,149.021
C08628=1216.805,-66.064,-38.829,179.740,5.402,149.021
C08629=1216.799,-65.815,-38.840,179.743,5.402,149.020
C08630=1216.794,-65.565,-38.851,179.745,5.402,149.019
C08631=1216.789,-65.316,-38.863,179.747,5.403,149.019
C08632=1216.784,-65.066,-38.875,179.749,5.402,149.018
C08633=1216.779,-64.816,-38.886,179.752,5.403,149.017
C08634=1216.774,-64.566,-38.898,179.755,5.403,149.017
C08635=1216.769,-64.316,-38.910,179.757,5.403,149.016
C08636=1216.763,-64.067,-38.922,179.760,5.403,149.015
C08637=1216.758,-63.818,-38.933,179.762,5.403,149.015
C08638=1216.753,-63.568,-38.945,179.764,5.403,149.014
C08639=1216.747,-63.318,-38.957,179.767,5.404,149.013
C08640=1216.743,-63.069,-38.968,179.769,5.403,149.013
C08641=1216.737,-62.819,-38.980,179.772,5.404,149.012
C08642=1216.732,-62.569,-38.991,179.774,5.404,149.011
C08643=1216.727,-62.319,-39.003,179.777,5.404,149.010
C08644=1216.722,-62.070,-39.016,179.778,5.404,149.010
C08645=1216.717,-61.820,-39.027,179.781,5.405,149.009
C08646=1216.712,-61.570,-39.039,179.783,5.405,149.009
C08647=1216.706,-61.320,-39.051,179.786,5.405,149.008
C08648=1216.702,-61.071,-39.062,179.788,5.405,149.007
C08649=1216.696,-60.821,-39.074,179.790,5.405,149.006
C08650=1216.691,-60.572,-39.086,179.793,5.405,149.006
C08651=1216.686,-60.323,-39.098,179.796,5.406,149.005
C08652=1216.680,-60.073,-39.109,179.798,5.405,149.004
C08653=1216.675,-59.823,-39.121,179.800,5.406,149.004
C08654=1216.671,-59.574,-39.133,179.802,5.405,149.003
C08655=1216.665,-59.324,-39.145,179.805,5.406,149.002
C08656=1216.660,-59.074,-39.157,179.808,5.406,149.001
C08657=1216.655,-58.824,-39.168,179.810,5.406,149.001
C08658=1216.650,-58.575,-39.181,179.813,5.406,149.000
C08659=1216.644,-58.325,-39.193,179.814,5.407,149.000
C08660=1216.639,-58.075,-39.205,179.817,5.407,148.999
C08661=1216.634,-57.825,-39.216,179.819,5.407,148.998
C08662=1216.629,-57.576,-39.229,179.822,5.407,148.997
C08663=1216.624,-57.326,-39.241,179.824,5.408,148.997
C08664=1216.619,-57.076,-39.252,179.826,5.407,148.996
C08665=1216.614,-56.827,-39.264,179.829,5.408,148.995
C08666=1216.609,-56.577,-39.276,179.831,5.407,148.995
C08667=1216.603,-56.327,-39.288,179.834,5.408,148.994
C08668=1216.599,-56.078,-39.300,179.836,5.408,148.993
C08669=1216.593,-55.828,-39.312,179.838,5.408,148.993
C08670=1216.588,-55.578,-39.324,179.841,5.408,148.992
C08671=1216.583,-55.329,-39.337,179.843,5.408,148.991
C08672=1216.577,-55.079,-39.348,179.846,5.409,148.990
C08673=1216.573,-54.829,-39.360,179.849,5.409,148.990
C08674=1216.568,-54.580,-39.372,179.850,5.409,148.989
C08675=1216.562,-54.330,-39.384,179.853,5.409,148.989
C08676=1216.557,-54.080,-39.396,179.856,5.410,148.988
C08677=1216.552,-53.831,-39.409,179.858,5.410,148.987
C08678=1216.547,-53.581,-39.420,179.860,5.410,148.986
C08679=1216.542,-53.332,-39.433,179.862,5.410,148.986
C08680=1216.536,-53.082,-39.445,179.865,5.410,148.985
C08681=1216.531,-52.833,-39.457,179.868,5.411,148.984
C08682=1216.526,-52.583,-39.469,179.870,5.410,148.984
C08683=1216.521,-52.333,-39.480,179.872,5.411,148.983
C08684=1216.517,-52.083,-39.493,179.874,5.410,148.982
C08685=1216.511,-51.833,-39.505,179.877,5.411,148.982
C08686=1216.506,-51.584,-39.518,179.880,5.411,148.981
C08687=1216.501,-51.334,-39.530,179.882,5.411,148.980
C08688=1216.495,-51.085,-39.542,179.885,5.411,148.979
C08689=1216.490,-50.835,-39.554,179.887,5.411,148.979
C08690=1216.485,-50.585,-39.567,179.889,5.412,148.978
C08691=1216.480,-50.336,-39.578,179.892,5.412,148.978
C08692=1216.475,-50.087,-39.591,179.894,5.412,148.977
C08693=1216.470,-49.837,-39.602,179.896,5.413,148.976
C08694=1216.464,-49.587,-39.615,179.899,5.413,148.975
C08695=1216.459,-49.337,-39.627,179.901,5.413,148.975
C08696=1216.454,-49.068,-39.641,179.904,5.413,148.974
C08697=1216.449,-48.797,-39.654,179.907,5.413,148.973
C08698=1216.442,-48.527,-39.667,179.909,5.413,148.972
C08699=1216.437,-48.258,-39.681,179.912,5.413,148.972
C08700=1216.432,-48.008,-39.692,179.914,5.414,148.971
C08701=1216.427,-47.758,-39.705,179.916,5.414,148.970
C08702=1216.421,-47.509,-39.718,179.919,5.414,148.970
C08703=1216.416,-47.259,-39.729,179.922,5.414,148.969
C08704=1216.411,-47.009,-39.742,179.924,5.414,148.968
C08705=1216.406,-46.759,-39.754,179.926,5.415,148.967
C08706=1216.401,-46.510,-39.767,179.929,5.415,148.967
C08707=1216.396,-46.260,-39.780,179.931,5.415,148.966
C08708=1216.391,-46.011,-39.791,179.933,5.416,148.966
C08709=1216.386,-45.762,-39.803,179.935,5.415,148.965
C08710=1216.381,-45.512,-39.815,179.938,5.416,148.964
C08711=1216.375,-45.262,-39.828,179.941,5.416,148.963
C08712=1216.371,-45.012,-39.841,179.943,5.416,148.963
C08713=1216.365,-44.762,-39.853,179.946,5.416,148.962
C08714=1216.360,-44.513,-39.865,179.948,5.417,148.961
C08715=1216.355,-44.264,-39.878,179.950,5.416,148.961
C08716=1216.350,-44.014,-39.890,179.953,5.417,148.960
C08717=1216.344,-43.764,-39.903,179.956,5.417,148.959
C08718=1216.339,-43.514,-39.916,179.958,5.417,148.959
C08719=1216.334,-43.265,-39.929,179.960,5.418,148.958
C08720=1216.329,-43.015,-39.940,179.962,5.417,148.957
C08721=1216.324,-42.766,-39.953,179.965,5.418,148.956
C08722=1216.319,-42.516,-39.966,179.968,5.418,148.956
C08723=1216.314,-42.266,-39.978,179.970,5.418,148.955
C08724=1216.309,-42.016,-39.991,179.972,5.418,148.954
C08725=1216.304,-41.767,-40.003,179.975,5.419,148.954
C08726=1216.298,-41.518,-40.016,179.977,5.419,148.953
C08727=1216.293,-41.268,-40.028,179.979,5.419,148.952
C08728=1216.288,-41.018,-40.041,179.982,5.420,148.952
C08729=1216.283,-40.768,-40.053,179.984,5.419,148.951
C08730=1216.278,-40.519,-40.066,179.987,5.420,148.950
C08731=1216.273,-40.270,-40.078,179.989,5.420,148.950
C08732=1216.268,-40.020,-40.090,179.992,5.420,148.949
C08733=1216.262,-39.769,-40.104,179.994,5.421,148.948
C08734=1216.257,-39.520,-40.116,179.997,5.421,148.948
C08735=1216.252,-39.271,-40.129,179.999,5.421,148.947
C08736=1216.247,-39.021,-40.142,-179.998,5.421,148.946
C08737=1216.242,-38.771,-40.154,-179.996,5.421,148.945
C08738=1216.237,-38.522,-40.166,-179.994,5.421,148.945
C08739=1216.232,-38.272,-40.179,-179.991,5.422,148.944
C08740=1216.227,-38.023,-40.192,-179.989,5.421,148.943
C08741=1216.222,-37.773,-40.205,-179.986,5.422,148.943
C08742=1216.216,-37.523,-40.218,-179.984,5.422,148.942
C08743=1216.211,-37.274,-40.230,-179.981,5.422,148.941
C08744=1216.206,-37.025,-40.243,-179.979,5.423,148.941
C08745=1216.201,-36.774,-40.255,-179.977,5.423,148.940
C08746=1216.196,-36.525,-40.268,-179.975,5.423,148.939
C08747=1216.190,-36.275,-40.281,-179.972,5.424,148.939
C08748=1216.185,-36.026,-40.294,-179.969,5.424,148.938
C08749=1216.181,-35.776,-40.307,-179.967,5.424,148.937
C08750=1216.176,-35.526,-40.319,-179.964,5.424,148.937
C08751=1216.170,-35.277,-40.332,-179.962,5.425,148.936
C08752=1216.165,-35.027,-40.345,-179.960,5.424,148.935
C08753=1216.160,-34.777,-40.358,-179.957,5.425,148.935
C08754=1216.155,-34.528,-40.371,-179.954,5.425,148.934
C08755=1216.150,-34.279,-40.383,-179.952,5.425,148.933
C08756=1216.145,-34.028,-40.397,-179.950,5.426,148.932
C08757=1216.139,-33.779,-40.409,-179.947,5.426,148.932
C08758=1216.134,-33.530,-40.422,-179.945,5.426,148.931
C08759=1216.130,-33.280,-40.435,-179.942,5.426,148.930
C08760=1216.124,-33.030,-40.448,-179.940,5.427,148.930
C08761=1216.119,-32.781,-40.461,-179.938,5.426,148.929
C08762=1216.114,-32.531,-40.474,-179.935,5.427,148.928
C08763=1216.109,-32.281,-40.486,-179.933,5.428,148.928
C08764=1216.103,-32.032,-40.500,-179.931,5.427,148.927
C08765=1216.099,-31.782,-40.513,-179.928,5.428,148.926
C08766=1216.094,-31.533,-40.525,-179.925,5.428,148.926
C08767=1216.089,-31.283,-40.538,-179.923,5.428,148.925
C08768=1216.083,-31.033,-40.551,-179.921,5.428,148.924
C08769=1216.078,-30.784,-40.564,-179.918,5.429,148.924
C08770=1216.073,-30.534,-40.576,-179.915,5.429,148.923
C08771=1216.068,-30.284,-40.590,-179.913,5.429,148.922
C08772=1216.063,-30.035,-40.603,-179.910,5.430,148.921
C08773=1216.058,-29.785,-40.616,-179.908,5.430,148.921
C08774=1216.053,-29.536,-40.630,-179.906,5.430,148.920
C08775=1216.047,-29.286,-40.642,-179.903,5.430,148.919
C08776=1216.043,-29.036,-40.655,-179.900,5.431,148.919
C08777=1216.037,-28.787,-40.668,-179.898,5.430,148.918
C08778=1216.032,-28.537,-40.681,-179.896,5.431,148.917
C08779=1216.027,-28.287,-40.694,-179.893,5.431,148.917
C08780=1216.022,-28.038,-40.707,-179.891,5.431,148.916
C08781=1216.017,-27.788,-40.721,-179.889,5.432,148.915
C08782=1216.012,-27.539,-40.733,-179.886,5.432,148.915
C08783=1216.006,-27.289,-40.747,-179.884,5.432,148.914
C08784=1216.002,-27.039,-40.759,-179.881,5.433,148.913
C08785=1215.997,-26.790,-40.772,-179.879,5.433,148.913
C08786=1215.992,-26.540,-40.786,-179.876,5.434,148.912
C08787=1215.987,-26.291,-40.799,-179.874,5.433,148.911
C08788=1215.981,-26.041,-40.812,-179.871,5.434,148.911
C08789=1215.976,-25.791,-40.825,-179.869,5.434,148.910
C08790=1215.971,-25.542,-40.838,-179.867,5.434,148.909
C08791=1215.966,-25.292,-40.852,-179.864,5.434,148.908
C08792=1215.961,-25.043,-40.865,-179.861,5.435,148.908
C08793=1215.956,-24.793,-40.878,-179.859,5.435,148.907
C08794=1215.951,-24.543,-40.891,-179.857,5.435,148.906
C08795=1215.946,-24.294,-40.905,-179.854,5.435,148.906
C08796=1215.941,-24.044,-40.918,-179.851,5.436,148.905
C08797=1215.935,-23.795,-40.930,-179.849,5.436,148.904
C08798=1215.931,-23.545,-40.945,-179.846,5.436,148.904
C08799=1215.925,-23.296,-40.957,-179.844,5.437,148.903
C08800=1215.920,-23.026,-40.971,-179.842,5.436,148.902
C08801=1215.914,-22.756,-40.986,-179.839,5.437,148.902
C08802=1215.909,-22.487,-41.000,-179.836,5.437,148.901
C08803=1215.903,-22.218,-41.015,-179.834,5.438,148.900
C08804=1215.899,-21.968,-41.028,-179.831,5.438,148.899
C08805=1215.893,-21.719,-41.042,-179.829,5.438,148.899
C08806=1215.889,-21.469,-41.055,-179.826,5.438,148.898
C08807=1215.883,-21.219,-41.068,-179.824,5.439,148.897
C08808=1215.879,-20.970,-41.081,-179.821,5.439,148.897
C08809=1215.873,-20.720,-41.095,-179.819,5.439,148.896
C08810=1215.868,-20.470,-41.108,-179.816,5.440,148.895
C08811=1215.863,-20.221,-41.121,-179.814,5.440,148.895
C08812=1215.857,-19.971,-41.135,-179.812,5.440,148.894
C08813=1215.852,-19.722,-41.148,-179.809,5.440,148.893
C08814=1215.847,-19.472,-41.162,-179.806,5.441,148.892
C08815=1215.842,-19.223,-41.175,-179.804,5.441,148.892
C08816=1215.837,-18.973,-41.189,-179.801,5.441,148.891
C08817=1215.832,-18.724,-41.201,-179.799,5.442,148.891
C08818=1215.827,-18.474,-41.216,-179.797,5.442,148.890
C08819=1215.822,-18.225,-41.228,-179.795,5.442,148.889
C08820=1215.817,-17.975,-41.243,-179.792,5.442,148.889
C08821=1215.811,-17.725,-41.256,-179.789,5.443,148.888
C08822=1215.807,-17.476,-41.269,-179.787,5.443,148.887
C08823=1215.801,-17.226,-41.283,-179.785,5.443,148.886
C08824=1215.797,-16.977,-41.296,-179.782,5.444,148.886
C08825=1215.791,-16.727,-41.310,-179.779,5.444,148.885
C08826=1215.786,-16.477,-41.324,-179.777,5.445,148.884
C08827=1215.781,-16.227,-41.337,-179.774,5.444,148.884
C08828=1215.776,-15.978,-41.351,-179.772,5.445,148.883
C08829=1215.771,-15.728,-41.364,-179.769,5.445,148.882
C08830=1215.766,-15.479,-41.378,-179.766,5.446,148.882
C08831=1215.761,-15.229,-41.391,-179.764,5.446,148.881
C08832=1215.756,-14.980,-41.404,-179.762,5.446,148.880
C08833=1215.751,-14.730,-41.418,-179.759,5.447,148.880
C08834=1215.746,-14.480,-41.432,-179.758,5.447,148.879
C08835=1215.741,-14.232,-41.446,-179.755,5.447,148.878
C08836=1215.735,-13.981,-41.459,-179.752,5.448,148.878
C08837=1215.730,-13.732,-41.473,-179.750,5.448,148.877
C08838=1215.725,-13.482,-41.486,-179.747,5.448,148.876
C08839=1215.720,-13.233,-41.500,-179.745,5.448,148.876
C08840=1215.715,-12.984,-41.514,-179.742,5.449,148.875
C08841=1215.710,-12.734,-41.527,-179.739,5.449,148.874
C08842=1215.705,-12.485,-41.541,-179.737,5.449,148.873
C08843=1215.700,-12.234,-41.555,-179.735,5.449,148.873
C08844=1215.695,-11.985,-41.568,-179.732,5.450,148.872
C08845=1215.690,-11.736,-41.582,-179.729,5.450,148.871
C08846=1215.685,-11.485,-41.596,-179.727,5.450,148.871
C08847=1215.680,-11.236,-41.610,-179.725,5.451,148.870
C08848=1215.675,-10.987,-41.623,-179.722,5.451,148.869
C08849=1215.669,-10.737,-41.637,-179.719,5.452,148.869
C08850=1215.664,-10.488,-41.651,-179.718,5.452,148.868
C08851=1215.660,-10.238,-41.665,-179.715,5.452,148.867
C08852=1215.655,-9.989,-41.679,-179.712,5.453,148.867
C08853=1215.649,-9.739,-41.692,-179.710,5.453,148.866
C08854=1215.644,-9.489,-41.706,-179.708,5.453,148.865
C08855=1215.639,-9.240,-41.721,-179.705,5.453,148.865
C08856=1215.634,-8.990,-41.733,-179.702,5.454,148.864
C08857=1215.629,-8.741,-41.747,-179.700,5.454,148.863
C08858=1215.624,-8.491,-41.762,-179.698,5.454,148.863
C08859=1215.618,-8.242,-41.776,-179.695,5.455,148.862
C08860=1215.614,-7.992,-41.789,-179.692,5.455,148.861
C08861=1215.609,-7.742,-41.803,-179.690,5.456,148.861
C08862=1215.604,-7.492,-41.817,-179.687,5.456,148.860
C08863=1215.598,-7.243,-41.831,-179.685,5.456,148.859
C08864=1215.593,-6.994,-41.845,-179.682,5.456,148.859
C08865=1215.589,-6.744,-41.858,-179.680,5.457,148.858
C08866=1215.583,-6.495,-41.872,-179.678,5.458,148.857
C08867=1215.578,-6.245,-41.887,-179.675,5.457,148.857
C08868=1215.573,-5.995,-41.901,-179.673,5.458,148.856
C08869=1215.568,-5.746,-41.915,-179.670,5.458,148.855
C08870=1215.563,-5.496,-41.929,-179.668,5.459,148.855
C08871=1215.558,-5.246,-41.942,-179.665,5.459,148.854
C08872=1215.553,-4.997,-41.956,-179.663,5.459,148.853
C08873=1215.548,-4.748,-41.970,-179.660,5.460,148.853
C08874=1215.543,-4.498,-41.984,-179.657,5.460,148.852
C08875=1215.538,-4.248,-41.999,-179.655,5.461,148.851
C08876=1215.533,-3.999,-42.013,-179.653,5.460,148.850
C08877=1215.528,-3.750,-42.027,-179.650,5.461,148.850
C08878=1215.523,-3.500,-42.041,-179.647,5.461,148.849
C08879=1215.518,-3.250,-42.055,-179.645,5.462,148.849
C08880=1215.513,-3.001,-42.069,-179.643,5.462,148.848
C08881=1215.508,-2.751,-42.082,-179.641,5.462,148.847
C08882=1215.503,-2.501,-42.097,-179.638,5.463,148.847
C08883=1215.498,-2.252,-42.111,-179.635,5.463,148.846
C08884=1215.493,-2.002,-42.125,-179.633,5.464,148.845
C08885=1215.487,-1.753,-42.139,-179.631,5.464,148.844
C08886=1215.482,-1.503,-42.153,-179.628,5.464,148.844
C08887=1215.477,-1.254,-42.168,-179.625,5.465,148.843
C08888=1215.472,-1.004,-42.182,-179.623,5.465,148.842
C08889=1215.467,-0.755,-42.196,-179.620,5.466,148.842
C08890=1215.462,-0.505,-42.210,-179.618,5.465,148.841
C08891=1215.457,-0.255,-42.224,-179.615,5.466,148.840
C08892=1215.452,-0.006,-42.239,-179.613,5.466,148.840
C08893=1215.447,0.244,-42.253,-179.610,5.467,148.839
C08894=1215.441,0.493,-42.267,-179.608,5.467,148.838
C08895=1215.436,0.743,-42.281,-179.606,5.467,148.838
C08896=1215.431,0.992,-42.295,-179.603,5.468,148.837
C08897=1215.426,1.242,-42.310,-179.600,5.468,148.836
C08898=1215.421,1.492,-42.324,-179.598,5.469,148.836
C08899=1215.416,1.740,-42.339,-179.596,5.469,148.835
C08900=1215.411,1.990,-42.353,-179.593,5.469,148.834
C08901=1215.406,2.240,-42.367,-179.590,5.470,148.834
C08902=1215.401,2.489,-42.381,-179.588,5.470,148.833
C08903=1215.396,2.739,-42.396,-179.585,5.471,148.832
C08904=1215.391,3.008,-42.411,-179.582,5.471,148.832
C08905=1215.386,3.277,-42.426,-179.580,5.472,148.831
C08906=1215.380,3.545,-42.442,-179.577,5.472,148.830
C08907=1215.375,3.815,-42.457,-179.574,5.473,148.830
C08908=1215.370,4.064,-42.471,-179.572,5.472,148.829
C08909=1215.365,4.314,-42.486,-179.570,5.473,148.828
C08910=1215.360,4.563,-42.500,-179.567,5.474,148.827
C08911=1215.355,4.813,-42.515,-179.564,5.474,148.827
C08912=1215.349,5.063,-42.529,-179.562,5.475,148.826
C08913=1215.344,5.312,-42.543,-179.560,5.474,148.825
C08914=1215.339,5.561,-42.558,-179.557,5.475,148.825
C08915=1215.334,5.811,-42.573,-179.554,5.475,148.824
C08916=1215.329,6.061,-42.587,-179.552,5.476,148.824
C08917=1215.324,6.310,-42.601,-179.549,5.477,148.823
C08918=1215.319,6.560,-42.615,-179.547,5.476,148.822
C08919=1215.315,6.809,-42.630,-179.545,5.477,148.822
C08920=1215.310,7.059,-42.645,-179.542,5.477,148.821
C08921=1215.304,7.309,-42.660,-179.539,5.478,148.820
C08922=1215.299,7.558,-42.673,-179.537,5.478,148.819
C08923=1215.294,7.807,-42.688,-179.534,5.479,148.819
C08924=1215.289,8.057,-42.703,-179.532,5.479,148.818
C08925=1215.284,8.306,-42.717,-179.529,5.479,148.817
C08926=1215.279,8.555,-42.732,-179.527,5.480,148.817
C08927=1215.274,8.805,-42.746,-179.524,5.480,148.816
C08928=1215.269,9.055,-42.761,-179.522,5.481,148.816
C08929=1215.264,9.305,-42.775,-179.519,5.482,148.815
C08930=1215.259,9.554,-42.790,-179.517,5.481,148.814
C08931=1215.254,9.804,-42.805,-179.515,5.482,148.814
C08932=1215.249,10.053,-42.819,-179.512,5.482,148.813
C08933=1215.244,10.303,-42.835,-179.509,5.483,148.812
C08934=1215.239,10.552,-42.849,-179.507,5.483,148.811
C08935=1215.234,10.802,-42.863,-179.504,5.484,148.811
C08936=1215.229,11.051,-42.878,-179.502,5.484,148.810
C08937=1215.224,11.301,-42.892,-179.499,5.484,148.809
C08938=1215.219,11.550,-42.908,-179.497,5.485,148.809
C08939=1215.213,11.799,-42.922,-179.494,5.486,148.808
C08940=1215.208,12.049,-42.936,-179.492,5.486,148.808
C08941=1215.204,12.298,-42.951,-179.489,5.487,148.807
C08942=1215.198,12.548,-42.966,-179.487,5.486,148.806
C08943=1215.193,12.797,-42.981,-179.484,5.487,148.806
C08944=1215.189,13.047,-42.995,-179.482,5.487,148.805
C08945=1215.184,13.296,-43.010,-179.479,5.488,148.804
C08946=1215.178,13.546,-43.025,-179.476,5.488,148.803
C08947=1215.173,13.796,-43.039,-179.474,5.489,148.803
C08948=1215.169,14.045,-43.054,-179.472,5.490,148.802
C08949=1215.164,14.295,-43.069,-179.470,5.489,148.802
C08950=1215.158,14.544,-43.084,-179.467,5.490,148.801
C08951=1215.153,14.794,-43.099,-179.464,5.491,148.800
C08952=1215.149,15.043,-43.114,-179.462,5.491,148.800
C08953=1215.143,15.293,-43.128,-179.459,5.492,148.799
C08954=1215.138,15.542,-43.143,-179.456,5.492,148.798
C08955=1215.133,15.792,-43.158,-179.454,5.493,148.798
C08956=1215.129,16.042,-43.174,-179.452,5.492,148.797
C08957=1215.124,16.291,-43.188,-179.449,5.493,148.796
C08958=1215.119,16.541,-43.203,-179.447,5.494,148.796
C08959=1215.114,16.790,-43.219,-179.444,5.494,148.795
C08960=1215.109,17.040,-43.233,-179.442,5.495,148.794
C08961=1215.104,17.289,-43.248,-179.439,5.495,148.794
C08962=1215.098,17.539,-43.263,-179.436,5.496,148.793
C08963=1215.094,17.788,-43.278,-179.434,5.496,148.792
C08964=1215.088,18.038,-43.293,-179.432,5.496,148.792
C08965=1215.083,18.287,-43.308,-179.429,5.497,148.791
C08966=1215.079,18.536,-43.323,-179.426,5.497,148.790
C08967=1215.073,18.786,-43.337,-179.424,5.498,148.790
C08968=1215.068,19.035,-43.352,-179.421,5.499,148.789
C08969=1215.064,19.284,-43.367,-179.419,5.499,148.788
C08970=1215.058,19.534,-43.382,-179.416,5.500,148.788
C08971=1215.053,19.783,-43.397,-179.414,5.499,148.787
C08972=1215.048,20.034,-43.413,-179.411,5.500,148.786
C08973=1215.044,20.283,-43.427,-179.409,5.500,148.786
C08974=1215.038,20.533,-43.443,-179.406,5.501,148.785
C08975=1215.033,20.782,-43.458,-179.403,5.501,148.784
C08976=1215.029,21.031,-43.472,-179.401,5.502,148.784
C08977=1215.023,21.281,-43.488,-179.399,5.503,148.783
C08978=1215.019,21.530,-43.503,-179.396,5.503,148.783
C08979=1215.013,21.780,-43.518,-179.393,5.504,148.782
C08980=1215.008,22.029,-43.533,-179.391,5.504,148.781
C08981=1215.003,22.279,-43.549,-179.389,5.504,148.781
C08982=1214.999,22.528,-43.564,-179.386,5.505,148.780
C08983=1214.993,22.778,-43.579,-179.383,5.505,148.779
C08984=1214.988,23.027,-43.594,-179.381,5.506,148.778
C08985=1214.983,23.277,-43.609,-179.379,5.507,148.778
C08986=1214.978,23.526,-43.624,-179.376,5.507,148.777
C08987=1214.973,23.776,-43.639,-179.373,5.508,148.777
C08988=1214.969,24.026,-43.654,-179.371,5.508,148.776
C08989=1214.963,24.275,-43.670,-179.369,5.508,148.775
C08990=1214.959,24.524,-43.685,-179.366,5.508,148.775
C08991=1214.953,24.774,-43.701,-179.363,5.509,148.774
C08992=1214.948,25.023,-43.715,-179.361,5.510,148.773
C08993=1214.943,25.273,-43.730,-179.358,5.510,148.773
C08994=1214.939,25.522,-43.746,-179.356,5.511,148.772
C08995=1214.933,25.772,-43.761,-179.353,5.511,148.771
C08996=1214.928,26.021,-43.777,-179.351,5.512,148.771
C08997=1214.923,26.270,-43.792,-179.348,5.513,148.770
C08998=1214.918,26.520,-43.808,-179.345,5.513,148.769
C08999=1214.913,26.769,-43.822,-179.343,5.513,148.769
C09000=1214.908,27.020,-43.838,-179.341,5.513,148.768
C09001=1214.904,27.269,-43.853,-179.338,5.514,148.768
C09002=1214.898,27.518,-43.868,-179.336,5.515,148.767
C09003=1214.893,27.767,-43.884,-179.333,5.515,148.766
C09004=1214.888,28.017,-43.899,-179.330,5.516,148.766
C09005=1214.883,28.267,-43.915,-179.328,5.516,148.765
C09006=1214.879,28.516,-43.930,-179.325,5.517,148.764
C09007=1214.873,28.765,-43.945,-179.323,5.517,148.764
C09008=1214.867,29.034,-43.962,-179.320,5.518,148.763
C09009=1214.863,29.302,-43.978,-179.317,5.518,148.762
C09010=1214.857,29.571,-43.995,-179.315,5.519,148.762
C09011=1214.852,29.841,-44.012,-179.312,5.520,148.761
C09012=1214.847,30.090,-44.027,-179.309,5.520,148.760
C09013=1214.842,30.339,-44.042,-179.307,5.521,148.759
C09014=1214.836,30.589,-44.058,-179.304,5.521,148.759
C09015=1214.832,30.838,-44.073,-179.302,5.522,148.758
C09016=1214.827,31.088,-44.089,-179.299,5.523,148.758
C09017=1214.822,31.337,-44.105,-179.297,5.523,148.757
C09018=1214.817,31.586,-44.120,-179.294,5.524,148.756
C09019=1214.812,31.836,-44.136,-179.292,5.523,148.756
C09020=1214.807,32.085,-44.152,-179.289,5.524,148.755
C09021=1214.802,32.335,-44.167,-179.287,5.524,148.754
C09022=1214.797,32.584,-44.182,-179.284,5.525,148.754
C09023=1214.792,32.834,-44.198,-179.282,5.526,148.753
C09024=1214.787,33.083,-44.214,-179.279,5.526,148.752
C09025=1214.782,33.332,-44.229,-179.276,5.527,148.752
C09026=1214.777,33.582,-44.245,-179.274,5.528,148.751
C09027=1214.772,33.832,-44.260,-179.271,5.528,148.750
C09028=1214.767,34.081,-44.276,-179.269,5.529,148.750
C09029=1214.763,34.331,-44.291,-179.266,5.529,148.749
C09030=1214.758,34.580,-44.308,-179.264,5.530,148.749
C09031=1214.752,34.829,-44.323,-179.261,5.531,148.748
C09032=1214.747,35.079,-44.339,-179.258,5.531,148.747
C09033=1214.743,35.328,-44.354,-179.256,5.532,148.747
C09034=1214.737,35.578,-44.370,-179.253,5.532,148.746
C09035=1214.732,35.827,-44.385,-179.251,5.533,148.746
C09036=1214.727,36.077,-44.402,-179.249,5.533,148.745
C09037=1214.722,36.326,-44.418,-179.246,5.533,148.744
C09038=1214.717,36.575,-44.433,-179.244,5.534,148.743
C09039=1214.713,36.825,-44.449,-179.241,5.534,148.743
C09040=1214.707,37.075,-44.464,-179.238,5.535,148.742
C09041=1214.702,37.323,-44.481,-179.236,5.536,148.741
C09042=1214.697,37.574,-44.496,-179.234,5.536,148.741
C09043=1214.692,37.823,-44.512,-179.231,5.537,148.740
C09044=1214.688,38.073,-44.527,-179.228,5.538,148.740
C09045=1214.683,38.321,-44.544,-179.226,5.538,148.739
C09046=1214.677,38.571,-44.559,-179.223,5.539,148.738
C09047=1214.673,38.821,-44.575,-179.220,5.539,148.738
C09048=1214.667,39.070,-44.591,-179.218,5.540,148.737
C09049=1214.662,39.319,-44.607,-179.216,5.541,148.737
C09050=1214.657,39.569,-44.623,-179.213,5.541,148.736
C09051=1214.653,39.818,-44.638,-179.210,5.542,148.735
C09052=1214.648,40.068,-44.655,-179.208,5.542,148.734
C09053=1214.643,40.317,-44.670,-179.205,5.543,148.734
C09054=1214.638,40.567,-44.686,-179.203,5.544,148.733
C09055=1214.633,40.816,-44.703,-179.200,5.544,148.733
C09056=1214.628,41.066,-44.718,-179.198,5.545,148.732
C09057=1214.623,41.316,-44.734,-179.195,5.545,148.731
C09058=1214.618,41.564,-44.750,-179.192,5.546,148.731
C09059=1214.612,41.814,-44.766,-179.190,5.546,148.730
C09060=1214.608,42.063,-44.783,-179.188,5.547,148.730
C09061=1214.603,42.313,-44.798,-179.185,5.548,148.729
C09062=1214.598,42.563,-44.814,-179.182,5.548,148.728
C09063=1214.593,42.812,-44.831,-179.180,5.549,148.728
C09064=1214.589,43.061,-44.846,-179.177,5.549,148.727
C09065=1214.584,43.310,-44.862,-179.175,5.550,148.726
C09066=1214.579,43.560,-44.878,-179.172,5.551,148.726
C09067=1214.574,43.809,-44.894,-179.170,5.551,148.725
C09068=1214.568,44.058,-44.910,-179.167,5.552,148.724
C09069=1214.564,44.309,-44.926,-179.164,5.553,148.724
C09070=1214.558,44.557,-44.942,-179.162,5.553,148.723
C09071=1214.554,44.807,-44.958,-179.160,5.554,148.723
C09072=1214.549,45.056,-44.975,-179.157,5.555,148.722
C09073=1214.544,45.306,-44.991,-179.154,5.555,148.721
C09074=1214.539,45.555,-45.007,-179.152,5.555,148.721
C09075=1214.534,45.805,-45.023,-179.150,5.555,148.720
C09076=1214.529,46.054,-45.039,-179.147,5.556,148.719
C09077=1214.524,46.304,-45.055,-179.145,5.557,148.719
C09078=1214.519,46.553,-45.071,-179.142,5.557,148.718
C09079=1214.514,46.803,-45.089,-179.139,5.558,148.717
C09080=1214.508,47.052,-45.104,-179.137,5.558,148.717
C09081=1214.504,47.302,-45.121,-179.134,5.560,148.716
C09082=1214.499,47.551,-45.136,-179.131,5.561,148.716
C09083=1214.494,47.800,-45.153,-179.129,5.561,148.715
C09084=1214.489,48.050,-45.169,-179.126,5.562,148.714
C09085=1214.484,48.299,-45.185,-179.124,5.562,148.714
C09086=1214.479,48.548,-45.202,-179.121,5.563,148.713
C09087=1214.474,48.798,-45.218,-179.119,5.564,148.713
C09088=1214.469,49.047,-45.234,-179.116,5.564,148.712
C09089=1214.465,49.297,-45.251,-179.113,5.565,148.711
C09090=1214.459,49.546,-45.266,-179.111,5.566,148.711
C09091=1214.455,49.795,-45.283,-179.108,5.566,148.710
C09092=1214.449,50.046,-45.299,-179.106,5.567,148.709
C09093=1214.444,50.295,-45.316,-179.103,5.568,148.709
C09094=1214.440,50.544,-45.332,-179.101,5.568,148.708
C09095=1214.434,50.794,-45.348,-179.098,5.569,148.707
C09096=1214.430,51.043,-45.365,-179.096,5.569,148.707
C09097=1214.425,51.292,-45.381,-179.093,5.570,148.706
C09098=1214.420,51.541,-45.398,-179.091,5.571,148.706
C09099=1214.415,51.792,-45.414,-179.088,5.571,148.705
C09100=1214.410,52.040,-45.430,-179.085,5.572,148.704
C09101=1214.405,52.290,-45.447,-179.083,5.572,148.704
C09102=1214.400,52.539,-45.463,-179.081,5.573,148.703
C09103=1214.395,52.789,-45.479,-179.078,5.574,148.703
C09104=1214.391,53.038,-45.496,-179.075,5.574,148.702
C09105=1214.385,53.287,-45.513,-179.073,5.575,148.701
C09106=1214.381,53.537,-45.530,-179.070,5.575,148.701
C09107=1214.375,53.786,-45.545,-179.068,5.576,148.700
C09108=1214.371,54.036,-45.562,-179.065,5.577,148.699
C09109=1214.366,54.286,-45.579,-179.063,5.577,148.699
C09110=1214.360,54.534,-45.595,-179.060,5.578,148.698
C09111=1214.356,54.784,-45.612,-179.057,5.579,148.697
C09112=1214.350,55.052,-45.629,-179.055,5.579,148.697
C09113=1214.345,55.321,-45.648,-179.052,5.581,148.696
C09114=1214.340,55.589,-45.666,-179.049,5.581,148.695
C09115=1214.335,55.858,-45.683,-179.046,5.582,148.695
C09116=1214.329,56.107,-45.700,-179.044,5.583,148.694
C09117=1214.325,56.357,-45.717,-179.042,5.583,148.694
C09118=1214.319,56.606,-45.733,-179.039,5.584,148.693
C09119=1214.315,56.855,-45.750,-179.036,5.584,148.692
C09120=1214.310,57.105,-45.767,-179.034,5.585,148.692
C09121=1214.305,57.354,-45.783,-179.032,5.586,148.691
C09122=1214.300,57.603,-45.800,-179.029,5.586,148.691
C09123=1214.295,57.854,-45.816,-179.026,5.587,148.690
C09124=1214.290,58.102,-45.833,-179.024,5.587,148.689
C09125=1214.285,58.352,-45.849,-179.021,5.589,148.689
C09126=1214.280,58.602,-45.867,-179.018,5.590,148.688
C09127=1214.275,58.850,-45.883,-179.016,5.590,148.687
C09128=1214.270,59.100,-45.900,-179.013,5.591,148.687
C09129=1214.265,59.350,-45.917,-179.011,5.592,148.686
C09130=1214.261,59.599,-45.933,-179.008,5.592,148.686
C09131=1214.256,59.848,-45.950,-179.006,5.593,148.685
C09132=1214.250,60.098,-45.967,-179.003,5.593,148.684
C09133=1214.246,60.347,-45.984,-179.001,5.594,148.684
C09134=1214.241,60.596,-46.000,-178.998,5.595,148.683
C09135=1214.236,60.846,-46.017,-178.996,5.595,148.683
C09136=1214.231,61.095,-46.034,-178.993,5.596,148.682
C09137=1214.226,61.345,-46.051,-178.991,5.597,148.682
C09138=1214.221,61.594,-46.067,-178.988,5.597,148.681
